    IF fRemDist < fPreTriggerPosition THEN
      eState             := cL_WAITSTART;
      tTrigger_EventTime := (tCurrentTime + LREAL_TO_ULINT(fRemDist / fI_ConveyorSpeed * 1E9));    // division save because we are moving to reach this position
      OnTriggerCommand   := cL_ACTIVE;  (*Arm EL2252*)

      LogTsDiff(aIdent := 'WAITALMOSTSTART: ', t1 := tTrigger_EventTime, t2 := tCurrentTime);
    ELSE
      eState           := cL_WAITALMOSTSTART;
      OnTriggerCommand := cL_INACTIVE;
    END_IF;

    ObTrigger := TRUE;

  cL_WAITSTART:       (*Wait until start time reached*)
    IF (tTrigger_EventTime < tCurrentTime) THEN (* StartTime elapsed *)
      // position reached
      eState           := cL_TRIGACTIVE;
      OnTriggerCommand := cL_INACTIVE; (*Disarm already command to EL2252, trigger generated*)
    ELSE
      // position not yet reached
      eState           := cL_WAITSTART;
      OnTriggerCommand := cL_ACTIVE;  (*Arm EL2252*)
    END_IF;

    ObTrigger := TRUE;  
    
  cL_TRIGACTIVE:   (*Trigger high*)
    eState := cL_WAITSTOP;
    
    // calculate end timestamp of trigger (end of trigger active signal)
    tTrigger_EventTime := (tTrigger_EventTime + LREAL_TO_ULINT(_fTriggerLength * 1E6));
    
    OnTriggerCommand := cL_INACTIVE;
    ObTrigger        := FALSE;
    
  cL_WAITSTOP:  (*Wait until trigger time has elapsed*)
    IF (tTrigger_EventTime < tCurrentTime) THEN (* StopTime elapsed *)
      eState           := cL_IDLE;
      OnTriggerCommand := cL_INACTIVE; (*Disarm EL2252, trigger generated*)
    ELSE
      eState           := cL_WAITSTOP;
      OnTriggerCommand := cL_ACTIVE;  (*Arm EL2252*)
    END_IF;

    ObTrigger        := FALSE;

  ELSE  (*Default*)
    eState           := cL_IDLE;
    ObTrigger        := FALSE;
    OnTriggerCommand := cL_INACTIVE;
END_CASE;

OtTriggerStartTime := tTrigger_EventTime;

(********************************* END OF FB *****************************************************)

METHOD Init
VAR_INPUT
  nResolution                   : LREAL := 1;      (*Printhead Resolution [e.g. 600] x Subpixel Resolution [e.g. 32]*)
  bUsePositionTrigger           : BOOL;            (*FALSE: Calculate time with speed and position distance@sensor evont*)
END_VAR
(*zero divisions*)
IF nResolution = 0 THEN RETURN; LogError('Invalid parameter'); END_IF;

// save config
_nResolution         := nResolution;
_bUsePositionTrigger := bUsePositionTrigger;

bInitOk := TRUE;
END_METHOD

(*
  Log timestamp difference (if verbose active).
  t1-t2 
*)
METHOD LogTsDiff : BOOL
VAR_INPUT
  aIdent : STRING;
  t1 : T_DCTIME64;
  t2 : T_DCTIME64;
END_VAR
IF _bVerbose THEN
  LogLvl(Lvl:=E_LogSeverity.Debug, Msg:=
       F_Concat7(aIdent, 
                 't1: ', TO_STRING(t1), 
                 ' t2: ', TO_STRING(t2), 
                 ' t1-t2 [ms]: ', TO_STRING((TO_LREAL(t1)-TO_LREAL(t2))*1E-6)
       )
  );
END_IF
END_METHOD

(*
  Detected start position X0 (absolute) in [SubPx].
*)
PROPERTY nStartPositionX0 : DINT
GET
nStartPositionX0 := _nX0;
END_GET
END_PROPERTY

PROPERTY UsePositionTrigger : BOOL
GET
UsePositionTrigger := _bUsePositionTrigger;
END_GET
SET
_bUsePositionTrigger := UsePositionTrigger;
END_SET
END_PROPERTY

END_FUNCTION_BLOCK

// ---- POUs/Products/FB_ModuleSynchronisation.TcPOU
FUNCTION_BLOCK FB_ModuleSynchronisation
VAR_INPUT
  IbEnable              : BOOL;             (*enable funcion*)
  IbEngaged             : ARRAY [1..iCPr_NB_PM] OF BOOL;
  IbPrintEnabled        : ARRAY [1..iCPr_NB_PM] OF BOOL;
  InFormatLength        : DINT;             (*format length [µm]*)
  InModule2ToModule3    : DINT;             (*distance between Module 2 and 3 [µm]*)
  IbFormatTrig          : BOOL;             (*format trigger*)
END_VAR

VAR_OUTPUT
  ObPrintEnabled        : ARRAY [1..iCPr_NB_PM] OF BOOL;
END_VAR

VAR
  fb_RFTrigPrintEnabled : RF_TRIG;
  fb_RTrigFormatTrig    : R_TRIG;
  _FormatTrigDelay      : DINT;             (*format trigger delay*)
  _FormatTrigCounter    : DINT;             (*format trigger counter*)
END_VAR

(*To start and stop printing of both modules synchronical the ObPrintEnabled of the second module must be delayed.*)
IF NOT IbEnable THEN
  ObPrintEnabled[1] := IbPrintEnabled[1];
  ObPrintEnabled[2] := IbPrintEnabled[2];
  RETURN;
END_IF

(*Trigger delay calculation*)
IF InFormatLength <> 0 THEN
  _FormatTrigDelay := InModule2ToModule3 / InFormatLength;
ELSE
  _FormatTrigDelay := 0;
END_IF

IF IbEngaged[1] THEN   (*Module2 active*)
  ObPrintEnabled[1] := IbPrintEnabled[1];   (*Module2 will print directly*)
  fb_RFTrigPrintEnabled(CLK := IbPrintEnabled[1]);
  IF fb_RFTrigPrintEnabled.RT THEN  (*Print start*)
    _FormatTrigCounter := 0;
    ObPrintEnabled[2] := FALSE;
  END_IF
  IF fb_RFTrigPrintEnabled.FT THEN  (*Print stop*)
    _FormatTrigCounter := 0;
  END_IF
  fb_RTrigFormatTrig(CLK := IbFormatTrig);
  IF fb_RTrigFormatTrig.Q THEN
    _FormatTrigCounter := _FormatTrigCounter + 1;
  END_IF
  IF _FormatTrigCounter >= _FormatTrigDelay THEN
    ObPrintEnabled[2] := IbPrintEnabled[2];     (*Module3 print is delayed*)
  END_IF
ELSE   (*Module3 can print directly*)
  ObPrintEnabled[1] := IbPrintEnabled[1];
  ObPrintEnabled[2] := IbPrintEnabled[2];
END_IF

END_FUNCTION_BLOCK

// ---- POUs/Products/obsolete/FB_CountWeu.TcPOU
FUNCTION_BLOCK FB_CountWeu
(*************************************************************************************************)
(*  FILENAME:    FB_CountWeu                                                                     *)
(*  PROJECT:     CALMAR PUPLC                                                                    *)
(*  COPYRIGHT:   All rights reserved (c) Wifag//Polytype, Fribourg/Switzerland (2021)            *)
(*  ENVIRONMENT: TwinCAT PLC                                                                     *)
(*  VERSION:     <version>                                                                       *)
(*************************************************************************************************)
(*  DESCRIPTION:                                                                   <description> *)
(*    Function for product count.                                                                *)
(*    The used pointers must be set in PRG_PRINT.Init!                                           *)
(*                                                                                </description> *)
(*************************************************************************************************)

VAR_INPUT
  pI_sAdsPrintUnit                          : POINTER TO ST_ADS_PU;        (*Pointer to ST_ADS_PU*)
  pI_ZeroPointerErr                         : POINTER TO UDINT;

  bI_SuccessFeedback                        : BOOL;             (*Success feedback from machine*)

  cI_ExtraCount                             : BYTE := 0;        (*Number of extra products that should be printed*)
END_VAR

VAR_OUTPUT
  bO_JobFinished                            : BOOL := FALSE;    (*Number of printed copies reached => job finished*)
  lO_ProductCountSuccess                    : UDINT;            (*Product counter of successfully printed*)
END_VAR

VAR
  iL_Counter                                : INT;              (*Local iteration counter - default*)

  lL_SuccessCount                           : UDINT := 0;       (*Success counter*)

  fb_RTrigSuccessFeedback                   : R_TRIG;           (*Success feedback from machine*)
  fb_RTrigPrintedCopies                     : R_TRIG;           (*Number of printed copies reached*)
END_VAR

(*0 pointer found*)
IF (pI_sAdsPrintUnit = 0) THEN
  IF pI_ZeroPointerErr <> 0 THEN
    pI_ZeroPointerErr^ := pI_ZeroPointerErr^ + 1;
  END_IF

  RETURN;
END_IF;

IF pI_sAdsPrintUnit^.sI_Start.bI_Command THEN
  lL_SuccessCount := 0;
END_IF;

(*Count successfull products*)
fb_RTrigSuccessFeedback(CLK := bI_SuccessFeedback);
IF fb_RTrigSuccessFeedback.Q THEN
  lL_SuccessCount := lL_SuccessCount + 1;
END_IF;
lO_ProductCountSuccess := lL_SuccessCount;

IF pI_sAdsPrintUnit^.sI_JobSettings.lI_NumberOfCopies = 0 THEN
  bO_JobFinished := FALSE;
ELSE
  (*Set job finished if number of desired copies reached.*)
  fb_RTrigPrintedCopies(CLK := (lL_SuccessCount >= (pI_sAdsPrintUnit^.sI_JobSettings.lI_NumberOfCopies + cI_ExtraCount)));
  IF fb_RTrigPrintedCopies.Q THEN
    bO_JobFinished := TRUE;
  END_IF;
END_IF;

(*Reset signals*)
IF pI_sAdsPrintUnit^.sI_Stop.bI_Command THEN
  bO_JobFinished := FALSE;
END_IF;

(********************************* END OF FB *****************************************************)

END_FUNCTION_BLOCK

// ---- POUs/Products/obsolete/FB_FIFO_DINT.TcPOU
FUNCTION_BLOCK FB_FIFO_DINT
(*************************************************************************************************)
(*  FILENAME:    FB_FIFO_TRIGGER_POS                                                             *)
(*  PROJECT:     CALMAR PUPLC                                                                    *)
(*  COPYRIGHT:   All rights reserved (c) Wifag//Polytype, Fribourg/Switzerland (2016)            *)
(*  ENVIRONMENT: TwinCAT PLC                                                                     *)
(*  VERSION:     <version>                                                                       *)
(*************************************************************************************************)
(*  DESCRIPTION:                                                                   <description> *)
(*    FIFO for trigger positions.                                                                *)
(*                                                                                </description> *)
(*************************************************************************************************)

{library public}
VAR_INPUT
  nI_FIFO_Input           : DINT;                          (*FIFO input value*)
  bI_Init                 : BOOL;                          (*Init*)
  bI_Add                  : BOOL;                          (*Add value*)
  bI_Release              : BOOL;                          (*Release value*)
END_VAR

VAR_OUTPUT
  bO_FIFO_Error           : BOOL;                          (*value FIFO error*)
  nO_FIFO                 : DINT;                          (*FIFO for value*)
END_VAR

{library private}
VAR
  nL_FIFO                 : ARRAY[0..iL_FIFOSIZE] OF DINT; (*FIFO for values*)
  iL_FIFO_Level           : INT := 0;                      (*Level of FIFO*)
  iL_Count                : INT;                           (*Temporary counter*)

  bL_Add                  : BOOL;                          (*Add value memory*)
  bL_Release              : BOOL;                          (*Release value memory*)
END_VAR

VAR CONSTANT
  (*Bit selection for configuration*)
  iL_FIFOSIZE             : INT := 75;
END_VAR

IF bI_Init THEN
  Init();
END_IF;

IF bI_Add AND NOT bL_Add THEN
  AddValue();
END_IF;
bL_Add := bI_Add;

IF bI_Release AND NOT bL_Release THEN
  ReleaseValue();
END_IF;
bL_Release := bI_Release;

nO_FIFO := nL_FIFO[0];
(********************************* END OF FB *****************************************************)

ACTION AddValue:
IF iL_FIFO_Level < iL_FIFOSIZE THEN
	nL_FIFO[iL_FIFO_Level] := nI_FIFO_Input;

	iL_FIFO_Level := iL_FIFO_Level + 1;
ELSE
	bO_FIFO_Error := TRUE;
END_IF;

(********************************* END OF ACTION *************************************************)
END_ACTION

ACTION Init:
iL_FIFO_Level := 0;
nL_FIFO[0]    := 0;
bO_FIFO_Error := FALSE;
(********************************* END OF ACTION *************************************************)
END_ACTION

ACTION ReleaseValue:
IF iL_FIFO_Level > 1 THEN
	FOR iL_Count := 0 TO (iL_FIFO_Level - 2) DO
		nL_FIFO[iL_Count] := nL_FIFO[iL_Count + 1];
	END_FOR;

	iL_FIFO_Level := iL_FIFO_Level - 1;
ELSIF iL_FIFO_Level = 1 THEN
	iL_FIFO_Level := 0;
END_IF;

(********************************* END OF ACTION *************************************************)
END_ACTION

END_FUNCTION_BLOCK

// ---- POUs/Products/obsolete/FB_HWLATCH.TcPOU
(* $Id$ *)
FUNCTION_BLOCK FB_HWLATCH
(*************************************************************************************************)
(*  FILENAME:     FB_HWLATCH.EXP			                                           		       		   *)
(*  PROJECT:      CALMAR PUPLC        																													 *)
(*  COPYRIGHT:    All rights reserved (c) Wifag//Polytype, Fribourg/Switzerland (2016)           *)
(*  ENVIRONMENT: 	TwinCAT PLC / CoDeSys																													 *)
(*	VERSION:			<version>																																			 *)
(*************************************************************************************************)
(*  DESCRIPTION:  Function block to convert hardware latch value [count] from terminal to print  *)
(*								system subpixel																																 *)
(*																																															 *)
(*************************************************************************************************)

{library public}
VAR_INPUT
	lI_Reference				:	UDINT;			(*position reference pulse count in [count]*)
	lI_Latch						:	UDINT;			(*position latch pulse count in [count]*)
	lI_Master_Position  :	DINT;				(*Current Master Position in [SubPx]*)
	fI_ResolutionInput	: LREAL:=1;	  (*Encoder Resolution in [um/increment]*)
	fI_ResolutionOutput	: LREAL:=1;	  (*Print system Resolution in [SubPx]*)
	bI_LatCVal					: BOOL;
	bI_Reset						: BOOL;				(*Reset terminal*)
END_VAR

VAR_OUTPUT
	iO_Offset_X0				: DINT;
	iO_Offset_XS				: DINT;
	bO_StartTrig				: BOOL;
	bO_EnLatC           : BOOL; 			(*C-Latch enable/reset @EL5101*)
END_VAR

{library private}
VAR
	lL_Latch_Reg				:	UDINT:=0;
  ll_Test             : UDINT:=0;
END_VAR

(*Latch register used for HW Start*)
IF lI_Latch <> lL_Latch_Reg AND bI_LatCVal THEN
  ll_Test := lI_Latch - lL_Latch_Reg;
	lL_Latch_Reg := lI_Latch;
	iO_Offset_X0 := lI_Master_Position - FC_LREAL_TO_DINT( (DINT_TO_LREAL(UDINT_TO_DINT(lI_Reference - lI_Latch)) * fI_ResolutionInput * (fI_ResolutionOutput / 25400) ));
	bO_StartTrig := TRUE;
ELSE
	bO_StartTrig := FALSE;
END_IF

(*Latch Handshake with Terminal EL5101,EnLatC must be set to 0 to reactivate latch input *)
IF bI_LatCVal THEN
	bO_EnLatC := FALSE;
ELSE
	bO_EnLatC := NOT bI_Reset;
END_IF

END_FUNCTION_BLOCK

// ---- POUs/Products/obsolete/FB_StartPositionDummy_HOA.TcPOU
(*
  A start position detection function block dummy.
  A dummy implementation to simulate start triggers at desired positions.
*)
FUNCTION_BLOCK FB_StartPositionDummy_HOA EXTENDS FB_BasePrint IMPLEMENTS I_StartPosDetect, I_PrintStatusClient, I_Simulation
VAR_INPUT
  bTrigger              AT%I* : BOOL;       // (INPUT) trigger (rising edge)
  tTrigger_TimeStamp    AT%I* : T_DCTIME64; // (INPUT) rigger timerstamp
  lPositionM2                 : DINT;       // current position [SubPx]
  fSpeedM2                    : LREAL;      // current speed [m/s]
  lPositionM3                 : DINT;       // current position [SubPx]
  fSpeedM3                    : LREAL;      // current speed [m/s]
  fResolution                 : LREAL;      // current print resolution [dpi*SubPx]
  nDelayTriggerDistance       : DINT;       // distance between CreateTrigger and DelayTrigger [SubPx]
  bMachineProdSpeed           : BOOL;       // machine reached production speed
  IpFormatLength              : POINTER TO DINT;  //pointer to format length if it's not used from iJobDefinition [µm]
END_VAR

VAR
  _bSim                 : BOOL;       // simulatio mode active (PROPERTY)
  _bCreateTrigger       : BOOL;       // create new CT trigger (PROPERTY)
  _nStartPosition       : DINT;       // create position for CT (absolut) [SubPx] (PROPERTY)
  _bCreateTriggerDelay  : BOOL;       // create delayed trigger (PROPERTY)
  _nDelayStartPosition  : DINT;       // create position for CT (absolut) [SubPx] (PROPERTY)
  fb_FIFOPositions      : FB_FIFO_DINT;
  _nFIFOPositionReg     : DINT;       // FIFO position register [SubPx]
  
  // local helper
  bNewCt              : BOOL;
  tCycle              : TIME;
  tonNewSheet         : TON;
  rfTrig_NewCT        : RF_TRIG;
  rfTrig_TriggerDelay : RF_TRIG;
  iJobDefinition      : CalmarCompPrint.I_JobDefinition;
  nCalcPosition       : DINT;            (*calculated position [SubPx]*)
  nCalcPositionM3     : DINT;            (*calculated position module 3 [SubPx]*)
  nDeltaPosition      : DINT;            (*delta position [SubPx]*)
  nDeltaPositionDelay : DINT;            (*delta position [SubPx]*)
  nSheetEndPosition   : DINT;            (*sheet end position [SubPx]*)
  nPositionRegM2      : DINT;            (*register position module 2 [SubPx]*)
  nPositionRegM3      : DINT;            (*register position module 3 [SubPx]*)
  nTriggerDistance    : DINT;            (*trigger distance [SubPx]*)
  bStartTrigger       : BOOL;            (*start trigger*)
  bSimStartTrigger    : BOOL;            (*simulated start trigger*)
  bSimStartActive     : BOOL;            (*simulated start active*)
  bInhibSensor        : BOOL;            (*inhibit sensor signals, TRUE=inhibit*)
  tCurrentTimeStamp   : T_DCTIME64;      (*get current timestamp*)
  fCurrentTimeStamp   : LREAL;           (*current timestamp*)
  fSensorTimeStamp    : LREAL;           (*sensor timestamp*)
  fDeltaDistance      : LREAL;           (*distance that the substrate moved between the detection and the treatment of the information [m]*)
END_VAR

VAR PERSISTENT
  // local simulation configurations persistent
  iCreateType    : UINT := 3;   // 0,1=by input rising edge, 2=create by sheets p.m. 3=create by sheet gap  
  fSheetCycle    : REAL := 20;  // [-] sheets per minute
  fSheetGap      : REAL := 0;   // [mm] gap between two sheets
  fSheetLength   : LREAL := 500; // [mm] sheet length TODO: remove if given by job(default if not given by jobDefinition)
END_VAR

VAR CONSTANT
  sCreateTArray : ARRAY[1..3] OF STRING := ['Input Trigger', 'Cycle', 'Gap'];
END_VAR

// Create CT triggers with a given cycle (based on configuration of Simulation)

(*If Module2 is disabled copy position from Module3*)
IF lPositionM2 = 0 THEN
  lPositionM2 := lPositionM3;
END_IF
(*Set nDelayTriggerDistance to minimum of 2 * IpFormatLength*)
IF (nDelayTriggerDistance <= LREAL_TO_DINT(F_SubPixelToMeter(2 * IpFormatLength^, fResSubPx := fResolution) * 1_000_000)) THEN 
  nDelayTriggerDistance := LREAL_TO_DINT(F_SubPixelToMeter(2 * IpFormatLength^, fResSubPx := fResolution) * 1_000_000);
END_IF


IF    iCreateType = 0 OR iCreateType = 1 OR NOT _bSim THEN   
  // --> trigger by input (default)
  IF bTrigger AND NOT bInhibSensor THEN
    bStartTrigger := TRUE;
    bInhibSensor  := TRUE;

    (* Calculate the current and sensor time stamp *)
    tCurrentTimeStamp := F_GetCurDcTaskTime64();
    fCurrentTimeStamp := (ULINT_TO_LREAL(tCurrentTimeStamp )) / 1_000_000.0; (*in ms*)
    fSensorTimeStamp  := fCurrentTimeStamp;// (ULINT_TO_LREAL(tTrigger_TimeStamp)) / 1_000_000.0; (*in ms*)
    (* Treatment of the information *)
    fDeltaDistance := (fCurrentTimeStamp - fSensorTimeStamp) * 0.001 * fSpeedM2;  (*Distance that the substrate moved between the detection and the treatment of the information [m]*)
    nCalcPosition     := lPositionM2 - F_MeterToSubPixel(fPosMeter := fDeltaDistance, fResoSubPx := fResolution);
    nSheetEndPosition := nCalcPosition + F_MeterToSubPixel(fPosMeter := fSheetLength / 1000, fResoSubPx := fResolution);
  ELSE
    bStartTrigger := FALSE;
	END_IF

  bNewCt := bStartTrigger;

ELSIF iCreateType = 2 AND _bSim THEN   
  // --> trigger by sheets per minute
  tCycle := prodspeed_to_time(lCycle := fSheetCycle);
  tonNewSheet(IN := NOT tonNewSheet.Q, PT := tCycle, Q => bNewCt);
  nCalcPosition := lPositionM2;
  
ELSIF iCreateType = 3 AND _bSim THEN
  // --> trigger by sheet gap;

  // fSheetLength from other source
  IF (IpFormatLength <> 0) THEN
    fSheetLength := DINT_TO_LREAL(IpFormatLength^) / 1000; // [µm] -> [mm]
  END_IF

  //  we need current job settings
  IF fSheetLength = 0 THEN fSheetLength := 1*1000; END_IF  // set some valid size 1000mm if no job is given
  (*trigger with timer is too inaccurate!*)
  (*
  IF (fSpeed > 0) THEN
    tCycle := length_to_time(dist := (fSheetGap + fSheetLength) / 1000, speed := fSpeed); 
    tonNewSheet(IN := NOT tonNewSheet.Q, PT := tCycle, Q => bNewCt);
  END_IF
  nCalcPosition := lPosition;
  *)

  (*trigger with distances*)
  bNewCt := FALSE;
  IF NOT bMachineProdSpeed THEN
    bSimStartActive  := FALSE;
  ELSE
    nTriggerDistance := F_MeterToSubPixel(fPosMeter := (fSheetGap + fSheetLength) / 1000, fResoSubPx := fResolution);

    IF NOT bSimStartActive THEN
      bSimStartActive     := TRUE;
      nDeltaPosition      := 0;
      nDeltaPositionDelay := 0;
      nPositionRegM2      := lPositionM2;
      nPositionRegM3      := lPositionM3;
		END_IF
    nDeltaPosition      := nDeltaPosition      + (lPositionM2 - nPositionRegM2);
    nDeltaPositionDelay := nDeltaPositionDelay + (lPositionM3 - nPositionRegM3);

    IF (nDeltaPosition >= nTriggerDistance) THEN
      bNewCt          := TRUE;
      nCalcPosition   := lPositionM2 - (nDeltaPosition - nTriggerDistance);
      nCalcPositionM3 := lPositionM3 - (nDeltaPosition - nTriggerDistance);
      nDeltaPosition  := nDeltaPosition - nTriggerDistance;
    END_IF
  END_IF
ELSE
  ;  // not supported ignore
END_IF


// Module 2: set ouputs (properties)
rfTrig_NewCT(CLK := bNewCt, RT => _bCreateTrigger);    // set ouput trigger
IF _bCreateTrigger THEN 
  _nStartPosition := nCalcPosition;
END_IF

// Module 3: set ouput for delay trigger (properties)
fb_FIFOPositions( bI_Init       := NOT bMachineProdSpeed  (*OR (nDelayTriggerDistance = 0)*)
                , bI_Add        := _bCreateTrigger
                , bI_Release    := _bCreateTriggerDelay
                , nI_FIFO_Input := nCalcPositionM3);
_nDelayStartPosition := fb_FIFOPositions.nO_FIFO + nDelayTriggerDistance;
IF _nFIFOPositionReg <> fb_FIFOPositions.nO_FIFO THEN
  nDeltaPositionDelay := (lPositionM3 - fb_FIFOPositions.nO_FIFO);
END_IF
_nFIFOPositionReg := fb_FIFOPositions.nO_FIFO;

rfTrig_TriggerDelay( CLK :=     (nDeltaPositionDelay >= nDelayTriggerDistance) 
                            AND bMachineProdSpeed
                            AND (fb_FIFOPositions.nO_FIFO <> 0)
                   , RT => _bCreateTriggerDelay);    // set ouput trigger


(*stop trigger to reset bInhibSensor*)
IF (lPositionM2 >= nSheetEndPosition) AND bInhibSensor THEN
  bInhibSensor := FALSE;
END_IF;

(*register position*)
nPositionRegM2 := lPositionM2;
nPositionRegM3 := lPositionM3;

PROPERTY bSimEnable : BOOL
GET
bSimEnable := _bSim;
END_GET
SET
_bSim := bSimEnable;
END_SET
END_PROPERTY

(*
  A new container detected.
  NOTE: a pulse only
*)
PROPERTY bStartTrig : BOOL
GET
bStartTrig := _bCreateTrigger;
END_GET
END_PROPERTY

(*
  A new container detected.
  NOTE: a pulse only
*)
PROPERTY bStartTrigDelay : BOOL
GET
bStartTrigDelay := _bCreateTriggerDelay;
END_GET
END_PROPERTY

(*
  A valid container detected.
*)
PROPERTY bValid : BOOL
GET
bValid := TRUE;
END_GET
END_PROPERTY

(*
Convert a distance to time with current speed
*)
METHOD PRIVATE length_to_time : TIME
VAR_INPUT
  dist  : LREAL; // [m] distance
  speed : LREAL; // [m/s] @speet
END_VAR
IF speed = 0 THEN  RETURN; END_IF   // ignore if speed = 0

length_to_time := LREAL_TO_TIME((dist * 1000)/ speed);  // TIME base is in [ms]
END_METHOD

METHOD mJobPause
END_METHOD

METHOD mJobStart
VAR_INPUT
	sJobDef	: CalmarCompPrint.I_JobDefinition;
END_VAR

// sample new CT configuration from job
iJobDefinition := sJobDef;    // current job definition

// fSheetLength from job definition
IF (iJobDefinition <> 0) AND (IpFormatLength = 0) THEN
  fSheetLength := iJobDefinition.fSubstrateDepth * 1000; // [m] -> [mm]
END_IF
// fSheetLength from other source
IF (IpFormatLength <> 0) THEN
  fSheetLength := DINT_TO_LREAL(IpFormatLength^) / 1000; // [µm] -> [mm]
END_IF

bInhibSensor := FALSE;
END_METHOD

METHOD mJobStop
VAR_INPUT
	sStatus	: CalmarCompPrint.I_JobStatus;
END_VAR
iJobDefinition := 0;    // delete job definition
END_METHOD

METHOD mProduced
VAR_INPUT
	(* current progress*)
	sProgress	: CalmarCompPrint.I_JobProgress;
END_VAR
; // nothing to do
END_METHOD

(*
  Detected start position X0 (absolute) in [SubPx].
*)
PROPERTY nDelayStartPositionX0 : DINT
GET
nDelayStartPositionX0 := _nDelayStartPosition;
END_GET
END_PROPERTY

(*
  Detected start position X0 (absolute) in [SubPx].
*)
PROPERTY nStartPositionX0 : DINT
GET
nStartPositionX0 := _nStartPosition;
END_GET
END_PROPERTY

(*
Convert production speed to a time. E.g. number of sheet per minute to a cycle time.
*)
METHOD PRIVATE prodspeed_to_time : TIME
VAR_INPUT
  lCycle        : REAL;    // sheets per minute
END_VAR
VAR
  fCycleTime    : LREAL;
END_VAR
fCycleTime := (60 / REAL_TO_LREAL(lCycle)) * 1000;
prodspeed_to_time := LREAL_TO_TIME(fCycleTime);
END_METHOD

METHOD reset
VAR_INPUT
END_VAR
bSimStartActive := FALSE;
END_METHOD

METHOD SimEnter : BOOL
LogInfo('Enter start position creator simulation');
_bSim := TRUE;
END_METHOD

METHOD SimExit : BOOL
LogInfo('Exit start position creator simulation');
_bSim := FALSE;
END_METHOD

METHOD SimUpdate : BOOL
; // nothing to do
END_METHOD

END_FUNCTION_BLOCK

// ---- POUs/Products/obsolete/FB_WorkerWeu.TcPOU
FUNCTION_BLOCK ABSTRACT FB_WorkerWeu EXTENDS FB_Worker
VAR_OUTPUT
  bError        : BOOL;       // an error is active
  nError        : UDINT;      // error code if error active, =0 else
END_VAR
VAR
  // config
  _pCtManager       : POINTER TO FB_CTManagerDefGrid;  // CT Manager reference
  _nTrackPosDomain  : E_PosDomain;    // Tracking position domain 
  _fPrintResolution : LREAL := 1;     // print(head) resolution in [dpi]
  _fSubPxResolution : LREAL := 1;     // SubPixel resolution [SubPx], resolution factor (fI_PrintResolution*fI_SubPxResolution=>Output resolution
  _name             : STRING;         // Worker name
  _sVisuName        : STRING := 'VISU_WorkerWeu'; // Worker visu instance name
  _pEcSrc           : POINTER TO T_ErrSrc;       // Error source definition

  // job
  _bJobActive       : BOOL;           // a job is active
  // ct
  _pAttachedCt      : POINTER TO FB_ContainerDefGrid;  // currently attached container
  fCtPosition       : LREAL;          // Container position relative to worker position in [SubPx (E_PosDomain.master_pos)]
  _bForceRelease    : BOOL;
END_VAR
VAR_STAT
  // static variables, same for all Workers
  _aJobName         : T_MaxString;
  _aJobGuid         : T_MaxString;
  _fImageWidthM     : LREAL;          // image width in [m]
  _fImageDepthM     : LREAL;          // image depth in [m]
  _fCtSecurityReleasePos : LREAL := 0;     // [SubPx] position where to release current ct at last (security release)
END_VAR
VAR PERSISTENT
  _fWorkerPosition  : LREAL;          // worker position relative to X0 in [m]
END_VAR

(*
  Generic abort implementation of DefGrid CT.
*)
METHOD Abort
VAR_INPUT
  iCT       : I_CT;
  sReason   : STRING;
END_VAR
VAR
  _pCt   : POINTER TO FB_ContainerWeu;
END_VAR
IF getCtInst(iCT:=iCT, pCT=>_pCt) <> 0 THEN  // get specific container
  // Do generic known aborts on CT
END_IF
END_METHOD

METHOD PROTECTED  Attach : BOOL
VAR_INPUT
  iCT       : I_CT;            (*container at triggered event position*)
END_VAR
VAR
  _pNewCt   : POINTER TO FB_ContainerWeu;

END_VAR
IF iCT = 0 THEN
  LogError(Msg:='attach failed -> not ct given');
  
ELSIF bEnable AND _pAttachedCt = 0 THEN           // enabled and free to attach
  IF getCtInst(iCT:=iCT, pCT=>_pNewCt) <> 0 THEN  // get specific container
    _pAttachedCt := _pNewCt;
    Attach:=TRUE;                                 // attach new
  ELSE
    LogError(Msg:='attach failed');
  END_IF
  
ELSIF bEnable AND _pAttachedCt <> 0 THEN    // enabled and already a CT attached
  LogError(Msg:='another container already attached -> ignore new (set error)');
  Abort(iCT:=iCT, sReason:='attach failed');  // abort new CT
    
ELSIF NOT bEnable AND _pAttachedCt <> 0 THEN // disabled and already a CT attached
  // force release if any hanging, and ignore attach
  Release(iCT:=_pAttachedCt^);

ELSIF NOT bEnable AND _pAttachedCt = 0 THEN  
  ;   // nothing to do, ignore attach

ELSE      // unspecified (error)case just log it
  LogError(Msg:='not tracked case');
END_IF
END_METHOD

{attribute 'monitoring':='call'}
PROPERTY bAttached : BOOL
GET
IF _pAttachedCt <> 0 THEN
  bAttached := TRUE;
END_IF
END_GET
END_PROPERTY

{attribute 'monitoring':='call'}
PROPERTY fPosition : LREAL
GET
fPosition := _fWorkerPosition;
END_GET
SET
_fWorkerPosition := fPosition;
setupPosition();
END_SET
END_PROPERTY

{attribute 'monitoring':='call'}
PROPERTY fPrintResolution : LREAL
GET
fPrintResolution := _fPrintResolution;
END_GET
SET
_fPrintResolution := fPrintResolution;
setupPosition();
END_SET
END_PROPERTY

(*
  Get specific container from interface.
  Returns specific container in return value and output parameter.
*)
METHOD INTERNAL getCtInst : POINTER TO FB_ContainerWeu
VAR_INPUT
  iCT              : I_CT;                         (*container at triggered event position*)
END_VAR
VAR_OUTPUT
  pCT              : POINTER TO FB_ContainerWeu;
END_VAR
pCT := 0;
IF _pCtManager <> 0 THEN
  getCtInst := _pCtManager^.GetContainerInstance(iCT);   // get real ct fb inst
  IF getCtInst <> 0 THEN
    pCT := getCtInst;   // OK all good
  ELSE
    LogError(Msg:='specific container not found');
	END_IF
ELSE
  LogError(Msg:='no container manager');
END_IF
END_METHOD

METHOD Init
VAR_INPUT
  pCtManager : POINTER TO FB_CTManagerWeu;       // CTManager
  fPrintResolution : LREAL := 1;                 // print(head) resolution in [dpi]
  fSubPxResolution : LREAL := 1;                 // SubPixel resolution [SubPx], resolution factor (fI_PrintResolution*fI_SubPxResolution=>Output resolution)
END_VAR
_pAttachedCt:=0;

IF pCtManager = 0 THEN
  LogError(Msg:='Init: invalid parameter');
  RETURN;
END_IF

// save config
_pCtManager := pCtManager; 
_fPrintResolution := fPrintResolution;
_fSubPxResolution := fSubPxResolution;
_fCtSecurityReleasePos := 0;
setupPosition();

setName('');

// register worker CTManager/Tracker event subject
_nTrackPosDomain := E_PosDomain.master_pos;
_pCtManager^.RegisterPosition(nPosDomain:=_nTrackPosDomain, iPositionEvent:=THIS^);

// init error source reference
_pEcSrc := ErrorCodes.fbErrCodeMngr.registerErrSource(
 nLocId := 0,
 aInstPath := InstanceName,
 aLocDescr := _name
);
IF _pEcSrc = 0 THEN LogError('could not register error source'); END_IF

bInitialized := TRUE;
END_METHOD

METHOD  ABSTRACT mJobStart
VAR_INPUT
	sJobDef	: CalmarCompPrint.I_JobDefinition;
END_VAR
END_METHOD

METHOD ABSTRACT mJobStop
VAR_INPUT
	sStatus	: CalmarCompPrint.I_JobStatus;
END_VAR
END_METHOD

(*
  Release CT from Worker.
  :return: TRUE if CT was released, FALSE if no CT was registered 
*)
METHOD Release : BOOL
VAR_INPUT
  iCT              : I_CT;                         (*container at triggered event position*)
END_VAR
IF iCT <> 0 AND _pAttachedCt <> 0 THEN Release := TRUE; END_IF
_pAttachedCt:=0;
END_METHOD

METHOD PRIVATE setName : BOOL
VAR_INPUT
  sName : STRING;
END_VAR
VAR
  nIdx : INT;
  bDone : BOOL;
END_VAR
IF sName = '' THEN
  // generate worker name
  _name := THIS^.InstanceName;
  WHILE NOT bDone DO
    nIdx := FIND(_name, '_');
    IF nIdx = 0 THEN bDone := TRUE; EXIT; 
    ELSE
      _name := RIGHT(_name,LEN(_name)-nIdx);
    END_IF 
  END_WHILE
ELSE
  _name := sName;  
END_IF
END_METHOD

METHOD PROTECTED setupPosition
_nTrackOffset := F_MeterToSubPixel(fPosMeter:=fPosition, fResoSubPx:=_fPrintResolution*_fSubPxResolution);
END_METHOD

METHOD  work
//Work only with attached container
IF _pAttachedCt <> 0 THEN 
  
  // update CT position
  fCtPosition := _pAttachedCt^.GetPos(nPosDomain:=E_PosDomain.master_pos) - _nTrackOffset; 

  // release CT (manually and security)
  IF _bForceRelease THEN
    LogWarning(F_Concat2('Manually realease CTId=', TO_STRING(_pAttachedCt^.pCT^.iId)));
    Release(iCT:=_pAttachedCt^);
  ELSIF _fCtSecurityReleasePos > 0 AND (fCtPosition > _fCtSecurityReleasePos) THEN
    LogError(F_Concat2('Security released CTId=', TO_STRING(_pAttachedCt^.pCT^.iId)));
    Release(iCT:=_pAttachedCt^);
  END_IF
  
END_IF
END_METHOD

END_FUNCTION_BLOCK

// ---- POUs/Products/obsolete/FB_WorkerWeu_Print.TcPOU
FUNCTION_BLOCK FB_WorkerWeu_Print EXTENDS FB_WorkerWeu
VAR_INPUT
  nEncoderPos   : DINT;       // Absolute print position [SubPx]
  fEncoderSpeed  : LREAL;     // Print speed [m/s]
  bHardwareSync : BOOL;
  bHardwareHold : BOOL;
  fPrintStartOffset : LREAL;  //PU->PG/PA offset
  fPrintYOffset : LREAL;      //Y-Shift in ram memory
END_VAR
VAR_OUTPUT
END_VAR
VAR
  fbPs              : FB_PS;
  fbPa              : FB_PA;
  fB_PcAdapter      : FB_PC_Adapter;
  
  _fPrintStartOffset : LREAL;   // internal print start offset
  _nPosX0            : DINT;    // X0 for last attached CT (detected postion)
  _nPosXS            : DINT;    // XS for last attached CT (shifted print start position)
  _nPosXDelta        : DINT;    // Shift value X0 -> XS
  _fPosY             : LREAL;    // Y shift for last attached CT
  _bPaStarted        : BOOL;
  _bPaStartRequested : BOOL;
  fBStartTimeout     : TON;
  rTrigSync          : R_TRIG;

  (*Messaging*)
  _bMsgInitialized   : BOOL;
  fb_MsgQueue        : FB_MSG_QUEUE;                        (*Message queue*)
  fb_MsgHandler      : FB_MSG_HANDLER;                      (*Message handler*)
  sL_MsgConfig       : ST_MSG_CONFIG;                       (*Message config*)
  fb_Msg             : ARRAY [1..iC_NUM_MSG] OF FB_MESSAGE; (*Messages*)
END_VAR
VAR PERSISTENT
  _fStartShiftOffset : LREAL := fC_START_SHIFT_OFFSET;
  _fStartShiftFactor : LREAL := fC_START_SHIFT_FACTOR;
END_VAR
VAR CONSTANT
  iC_NUM_MSG : UDINT := 5;
  fC_START_SHIFT_FACTOR : LREAL := -2.4E-2;
  fC_START_SHIFT_OFFSET : LREAL := -1.0E-2;
END_VAR


//TODO Add error/warnings
bError := FALSE;
nError := 0;

//Start offset update
IF _fPrintStartOffset <> fPrintStartOffset THEN //Worker position changed
  IF _pAttachedCt = 0 THEN //Update only without attached container
    _fPrintStartOffset :=fPrintStartOffset;
	END_IF
END_IF

//Worker position update
IF _fWorkerPosition <> (_fPrintStartOffset + (_fStartShiftOffset + _fStartShiftFactor * fEncoderSpeed))  THEN //Worker position changed (camera settings change)
  IF _pAttachedCt = 0 THEN //Update only without attached container
    // WorkerPosition
    fPosition := _fPrintStartOffset + (_fStartShiftOffset + _fStartShiftFactor * fEncoderSpeed);
	END_IF
END_IF

(*---- Messaging -----------------------*)
IF _bMsgInitialized THEN
  fb_MsgHandler();
  {warning 'TODO: implement PrintWorker & PG messages'}
  //fB_Msg[1](bI_Status := dfsdfdsf);
  fb_MsgQueue();
END_IF

PROPERTY aPaState : STRING
GET
aPaState := fbPa.aPaState;
END_GET
END_PROPERTY

METHOD PROTECTED  Attach : BOOL
VAR_INPUT
  iCT              : I_CT;                         (*container at triggered event position*)
END_VAR
Attach:=FALSE;

IF bEnable AND SUPER^.Attach(iCT:=iCT) THEN
  // Additional worker checks
    // - job is valid?
  IF _pAttachedCt^.pJob = 0 OR NOT _bJobActive THEN
    Release(iCT:=iCT);
    RETURN;   // do not print
  
  // CT valid & CT present
  ELSIF NOT _pAttachedCt^.bValid OR NOT _pAttachedCt^.bProductPresent THEN
    Release(iCT:=iCT);
    RETURN;   // do not print
  
  // Ignore start due to hardware hold  
  ELSIF bHardwareHold THEN
    //_pAttachedCt^.setError(ErrDef:=EC_Print.ecPaAbortHold, Src:=_pEcSrc^);
    Release(iCT:=iCT);
    RETURN;   // do not print
  // - OK attach
  ELSE
    Attach := TRUE;
	END_IF
  
  
  //Prepare print station
  fbPs.bPrintEnable := iCT.bValid AND iCT.bProductPresent;

  //Start print, PA should be in READY or DONE
  
  // Set X print position
  _nPosX0 := _pAttachedCt^.getPosX0(nPosDomain:=E_PosDomain.master_pos);
  _nPosXDelta := F_MeterToSubPixel(_fPrintStartOffset,_fPrintResolution*_fSubPxResolution); // + PG/PA Shift (additional PG offset 0 for firstLine)

  _nPosXS := _nPosX0 + _nPosXDelta;
  fB_PcAdapter.setPrintStartPos(nX0:=_nPosXS);
  
  // Set Y print position
  _fPosY := fPrintYOffset;
  fB_PcAdapter.setPrintYShift(nYShift:=FC_LREAL_TO_DINT(_fPosY));

  // check
  IF _nPosXS < nEncoderPos THEN
    LogWarning(Msg:='Print start position < Encoder position');
	END_IF
    
  IF fbPa.printStart() THEN
    _bPaStarted := FALSE;
    _bPaStartRequested := TRUE;
    Attach:=TRUE;
    LogLvl(Lvl:=E_LogSeverity.Debug, F_Concat2('printStart:', _pAttachedCt^.print(0)));  // print container
    LogLvl(Lvl:=E_LogSeverity.Debug, F_Concat4('> XS:', TO_STRING(_nPosXS), ' = X0:', TO_STRING(_pAttachedCt^.GetPosX0(nPosDomain:=E_PosDomain.master_pos))));
    LogLvl(Lvl:=E_LogSeverity.Debug, F_Concat2( ' + shStartOffs:', TO_STRING(F_MeterToSubPixel(_fPrintStartOffset,_fPrintResolution*_fSubPxResolution))));

  ELSE  
    LogError(Msg:='PA not ready to start at attach');
    Release(iCT := iCT);
	END_IF
  
ELSE
  // parent attach failed case
END_IF
END_METHOD

METHOD InitMsg : BOOL
VAR_INPUT
  pMsgInterface : POINTER TO ST_ADS_MSG_IF;
END_VAR
VAR
  nCtr : UDINT;
END_VAR
IF pMsgInterface = 0 THEN RETURN; END_IF

(*Messaging*)
sL_MsgConfig.bI_Enable       := TRUE;
sL_MsgConfig.pI_FbMsgHandler := ADR(fb_MsgHandler);
fb_MsgHandler.pI_MsgQueue    := ADR(fb_MsgQueue);
fb_MsgQueue.pI_MsgInterface  := pMsgInterface;
fb_MsgQueue.cI_MaxElement    := 6;

(*Messages*)
FOR nCtr := 1 TO iC_NUM_MSG DO
  fb_Msg[nCtr].pI_MsgConfig       := ADR(sL_MsgConfig);
  fb_Msg[nCtr].iI_MsgLocation     := 0;
END_FOR
//fb_Msg[1].iI_MsgNumber       := ;
// ...

_bMsgInitialized := TRUE;
END_METHOD

METHOD InitWorkerPrint : BOOL
VAR_INPUT
END_VAR
IF NOT bInitialized THEN LogError('Base Worker not initialized! call init() before'); RETURN; END_IF

// worker specific init

//Print Aggregate
fbPa.bSyncAfterDone := FALSE;
fbPa.init(iPcAdapter := fB_PcAdapter, iPsInterface:=fbPs);
END_METHOD

METHOD   mJobStart
VAR_INPUT
	sJobDef	: CalmarCompPrint.I_JobDefinition;
END_VAR
IF NOT bEnable THEN RETURN; END_IF  // only if enabled

fbPa.jobStart();

_bJobActive := TRUE;
END_METHOD

METHOD  mJobStop
VAR_INPUT
	sStatus	: CalmarCompPrint.I_JobStatus;
END_VAR
fbPa.jobStop();
_bJobActive := FALSE;
END_METHOD

METHOD registerPc : BOOL
VAR_INPUT
  iNewPC : I_PC;
END_VAR
registerPc := fB_PcAdapter.registerPc(iNewPC := iNewPC);
END_METHOD

METHOD registerPh : BOOL
VAR_INPUT
    iPH : I_PH;
END_VAR
//Attach head to print station
IF iPH <> 0 THEN
  fbPs.registerPh(iNewPh:=iPH);
END_IF
END_METHOD

PROPERTY sPcFlags : CalmarCompPrint.ST_PC_FLAGS
GET
sPcFlags := fB_PcAdapter.sPcFlags;
END_GET
END_PROPERTY

PROPERTY sPcState :  CalmarCompPrint.ST_PG_STATUS
GET
VAR
  sJobStatus : ST_JobProgress;
END_VAR
sPcState.bStartPrintCanEx := fBPa.bStartCanEx;
sPcState.bStartPrintExec  := fBPa.bStartExec;
sPcState.bStopPrintCanEx  := fBPa.bStopCanEx;
sPcState.bStopPrintExec   := fBPa.bStopExec;
sPcState.bPausePrintCanEx := FALSE;       // obsolete ???
sPcState.bPausePrintExec  := FALSE;       // obsolete ???
sPcState.bReady           := fB_PcAdapter.bAllReady OR fB_PcAdapter.bAllDone;
sPcState.bError           := fB_PcAdapter.bError;
sPcState.bPrinting        := fB_PcAdapter.bAllPrinting;
sPcState.bLoad            := fB_PcAdapter.bAllPreparing;
sPcState.bArmed           := fB_PcAdapter.bAllPrinting OR fB_PcAdapter.bAllReady OR fB_PcAdapter.bAllDone OR fB_PcAdapter.bAllPreparing;
sPcState.bEnabled         := bEnable;
sPcState.bStartStrb       := fBPa.bStartStrb;
sPcState.bPcEnabled       := fB_PcAdapter.bPcEnable;
sPcState.lProductCount    := 0;            // obsolete ???
sPcState.sJobStatus       := sJobStatus;   // obsolete ???
END_GET
END_PROPERTY

METHOD  work
IF NOT bEnable THEN RETURN; END_IF

SUPER^.work();

(*Update virtual encoder on all controller boards*)
fB_PcAdapter.setEncoderPos(nEncoderPos);
fB_PcAdapter();

(*Call print aggregate*)
rTrigSync(CLK:=bHardwareSync); 
IF rTrigSync.Q THEN fbPa.sync(); END_IF   // external sync
fbPa.bHold := bHardwareHold;              // external hw hold
fbPa();

fBStartTimeout(IN := _bPaStartRequested,PT := T#60MS);

IF _pAttachedCt <> 0 AND bEnable THEN // Work only with attached container
  // PA control
  IF bHardwareHold THEN   // _pAttachedCt^.bValid AND
    // abort during printing
    _pAttachedCt^.setError(ErrDef:=EC_Print.ecPaAbortHold, Src:=_pEcSrc^);
    Release(_pAttachedCt^);
    
  ELSIF _bPaStartRequested THEN
    IF fbPa.bPrinting THEN
      _bPaStarted := TRUE;
      _bPaStartRequested := FALSE;
    ELSIF fBStartTimeout.Q THEN //Stop print at timeout to make ready for next container
      _bPaStarted := FALSE;
      _bPaStartRequested := FALSE;
      fbPa.printStop();
      _pAttachedCt^.setError(ErrDef:=EC_Print.ecPaStartErr, Src:=_pEcSrc^);
      Release(_pAttachedCt^);
		END_IF
  ELSIF _bPaStarted THEN
    // Set Y print position
    _fPosY := fPrintYOffset;
    fB_PcAdapter.setPrintYShift(nYShift := FC_LREAL_TO_DINT(_fPosY));

    //Release container when print finished
    IF fbPa.bDone OR fbPa.bStop THEN
      _bPaStarted := FALSE;
      Release(_pAttachedCt^);
    (*ELSIF fbpa.bError THEN
      _pAttachedCt^.setError(ErrDef:=EC_Print.ecPaPrintErr, Ident:=0);
      Release(_pAttachedCt^);*)
    END_IF 
	END_IF
END_IF  

(*Logging config*)
fbPa.LogLevel := LogLevel;
fB_PcAdapter.LogLevel := LogLevel;
END_METHOD

END_FUNCTION_BLOCK

// ---- POUs/Products/Print_Weu/UV_LED_Modul/FB_UvLedModule.TcPOU
FUNCTION_BLOCK FB_UvLedModule EXTENDS FB_BasePrint IMPLEMENTS I_DeviceBase
VAR_INPUT
  IbReady                  AT%I* : BOOL;
END_VAR

VAR_OUTPUT
  ObEnableHigh             AT%Q* : BOOL;
  ObLowIntenseMode         AT%Q* : BOOL;
  ObDisableLeft            AT%Q* : BOOL;
  ObDisableRight           AT%Q* : BOOL;
  OnIntensitySetpoint      AT%Q* : WORD;  (*Setpoint for intensity control  [digit]*)
END_VAR

VAR
  _bActivate                     : BOOL;
  _sName                         : STRING := '';
  _StInkDefinition               : ST_INKDEFINITON;
END_VAR

VAR CONSTANT
  CnAnalogMinDigit               : DINT := 0;      (*Min value analog-output in digit*)
  CnAnalogMaxDigit               : DINT := 32767;  (*Max value analog-output in digit*)
  CnMinIntensitySetpoint         : DINT := 5;      (*Min setpoint for intensity control [%]*)
  CnMaxIntensitySetpoint         : DINT := 100;    (*Max setpoint for intensity control [%]*)
END_VAR

VAR PERSISTENT
  RbLowIntenseMode               : BOOL := FALSE;  (*Visu: set low intense mode*)
  RbDisableLeft                  : BOOL := FALSE;  (*Visu: disable left SLM*)
  RbDisableRight                 : BOOL := FALSE;  (*Visu: disable right SLM*)
  RnIntensitySetpoint            : DINT := 20;     (*Visu: setpoint for intensity control [%]*)
END_VAR

(*Set outputs*)
ObEnableHigh        := _bActivate;
ObLowIntenseMode    := RbLowIntenseMode;
ObDisableLeft       := RbDisableLeft;
ObDisableRight      := RbDisableRight;
OnIntensitySetpoint := DINT_TO_WORD(CnAnalogMaxDigit * RnIntensitySetpoint / 100);  (*Setpoint [digit]*)

METHOD mDisable : BOOL
_bActivate := FALSE;
END_METHOD

METHOD mEnable : BOOL
_bActivate := TRUE;
END_METHOD

{warning 'add property implementation'}
PROPERTY pActive : BOOL
GET
pActive := _bActivate;
END_GET
END_PROPERTY

{warning 'add property implementation'}
PROPERTY pErrorCode : INT
GET
END_GET
END_PROPERTY

PROPERTY pStInkDefinition : ST_INKDEFINITON
SET
_StInkDefinition := pStInkDefinition;
END_SET
END_PROPERTY

END_FUNCTION_BLOCK

// ---- Project Information/F_GetCompany.TcPOU
// This function has been automatically generated from the project information.
{attribute 'signature_flag' := '1073741824'}
{attribute 'TcGenerated'}
{attribute 'no-analysis'}
FUNCTION F_GetCompany : WSTRING
VAR_INPUT
	
END_VAR

F_GetCompany := "WIFAG-Polytype";

END_FUNCTION

// ---- Project Information/F_GetTitle.TcPOU
// This function has been automatically generated from the project information.
{attribute 'signature_flag' := '1073741824'}
{attribute 'TcGenerated'}
{attribute 'no-analysis'}
FUNCTION F_GetTitle : WSTRING
VAR_INPUT
	
END_VAR

F_GetTitle := "PUPLC";

END_FUNCTION

// ---- GlobalTextList.TcGTLO
TEXTLIST GlobalTextList
  469 = ' '
  412 = '  %d'
  419 = '  %s'
  415 = '  0x%X'
  585 = '  1     2    3     4    5     6    7    8'
  295 = '  :'
  13539 = '  > verbose Mode'
  10089 = '  Delta distance [m]: %f'
  818 = '  Dropspeed [m/s]: %f'
  13004 = '  Module for mark trigger: %d'
  16821 = '  Time distance [ms]: %d'
  782 = ' %f'
  7576 = ' %s'
  10973 = ' %s ID'
  10174 = ' (max %d)'
  24 = ' ActualLevel'
  2816 = ' Add. dead time [ms]: %f'
  476 = ' Base folder: %s'
  990 = ' Camera correction X [m]: %f'
  987 = ' Camera correction [m]: %f'
  781 = ' Camera offset Y [mm]: %f'
  772 = ' Camera position X [m]: %f'
  831 = ' Camera position [m]: %f'
  471 = ' CH0: %d %%'
  472 = ' CH1: %d %%'
  473 = ' CH2: %d %%'
  474 = ' CH3: %d %%'
  820 = ' Compensation [mm]: %f'
  828 = ' Current time stamp compensation [µs]: %d'
  489 = ' D: %d'
  4 = ' ErrorLevel'
  492 = ' FileNbrs : %d '
  493 = ' Files p. PC : %d '
  5911 = ' Head base plate gap to roller table [m]: %f'
  1154 = ' Head offset to base plate [m]: %f'
  484 = ' ID: %d'
  487 = ' JOB_ID: %d'
  805 = ' Mark Height Y [mm] : %f'
  804 = ' Mark Length X [mm] : %f'
  6067 = ' Offset [m]'
  986 = ' Offset [m] : %f'
  822 = ' Print Position [m]: %f'
  823 = ' Print Stop Position [m]: %f'
  228 = ' Progress: %d %%'
  491 = ' Resolution : %d '
  192 = ' Sel PH : %d '
  13302 = ' Select header tank : %d '
  978 = ' Select headertank : %d '
  11576 = ' Selected Balance : %d '
  517 = ' Selected BL : %d '
  168 = ' Selected Group : %d '
  79 = ' Selected PC : %d '
  85 = ' Selected PG : %d '
  18812 = ' Selected PH : %d '
  8193 = ' Selected PrintModule: %d '
  215 = ' Selected Unit : %d '
  920 = ' SelHeaderTank : %d '
  2 = ' SelStorTank : %d '
  821 = ' Sensor Position [m]: %f'
  829 = ' Sensor time stamp compensation [µs]: %d'
  776 = ' Sheet detect to camera [m]: %f'
  943 = ' Sheet detect to mark [mm]: %d'
  944 = ' Sheet detect to mark [m]: %d'
  945 = ' Sheet detect to mark [m]: %f'
  826 = ' Shift start correction [m] : %f'
  827 = ' Shift start offset [m] : %f'
  13811 = ' Speed-dependent factor [s]'
  985 = ' Speed-dependent factor [s] :\n %f'
  7284 = ' Substrate thickness [m]: %f'
  819 = ' Throw Distance [mm]: %f'
  778 = ' Trigger length [sec]: %f'
  488 = ' W: %d'
  3 = ' WarningLevel'
  194 = ' X: %s [um]'
  1900 = ' X: %s [µm]'
  200 = ' Y: %s [px]'
  4807 = '! Values not persisted\n  Testing only'
  5193 = '%.1f kg'
  1205 = '%.3f kg'
  4155 = '%.4f mV/V'
  4193 = '%0.01f'
  303 = '%0.0f'
  7 = '%0.0f [%%]'
  293 = '%0.1f'
  18487 = '%0.1f [m/min]'
  7779 = '%0.1f [mbar] '
  6147 = '%0.1f [um]'
  2166 = '%0.2f'
  16761 = '%0.2f [m/s]'
  993 = '%0.3f'
  6769 = '%0.3f [m/s]'
  13150 = '%0.3f [ms]'
  1141 = '%0.4f'
  397 = '%0.6f'
  4314 = '%0.6f [ms]'
  5810 = '%0.6f [m]'
  704 = '%1.1f'
  6 = '%1.1f l'
  1138 = '%1.1f mbar'
  679 = '%1.1f mm'
  675 = '%1.1f mm/s'
  907 = '%1.1f [mbar]'
  5754 = '%1.1f [mBar]'
  39 = '%1.1f [min]'
  1038 = '%1.1f [mm]'
  1528 = '%1.1f [ms]'
  905 = '%1.1f [°C]'
  26 = '%1.2f'
  10 = '%1.2f l'
  741 = '%1.2f mm'
  917 = '%1.2f [g/cm³]'
  19 = '%1.2f [kg/l]'
  7272 = '%1.2f [m/s]'
  916 = '%1.2f [mPa*s]'
  32 = '%1.3f'
  699 = '%1.3f mm'
  913 = '%1.3f [g/cm³]'
  2489 = '%1.3f [mm]'
  915 = '%1.3f [mPa*s]'
  14861 = '%1.4f'
  735 = '%1.4f m'
  9544 = '%1.4f mm'
  12078 = '%1.4f [mm]'
  2560 = '%1.4f [m]'
  702 = '%1.6f m'
  536 = '%2.3f'
  9 = '%d'
  956 = '%D'
  6010 = '%d '
  372 = '%d %%'
  11134 = '%d [%%]'
  909 = '%d [%]'
  6448 = '%d [0.01mm]'
  1357 = '%d [0.1%%]'
  6437 = '%d [0.1mm]'
  1034 = '%d [g/m2]'
  8223 = '%d [g/m^2]'
  1035 = '%d [m/min]'
  1043 = '%d [mbar]'
  2974 = '%d [mm]'
  21 = '%d [ms]'
  7034 = '%d [m]'
  3602 = '%d [px]'
  5286 = '%d [px] '
  911 = '%d [s]'
  1059 = '%d [°C]'
  1064 = '%d [µm]'
  365 = '%d%%'
  1307 = '%ds'
  456 = '%f'
  3157 = '%f [liter]'
  10485 = '%f [m/min]'
  5388 = '%f [mm]'
  812 = '%f [m]'
  2912 = '%f [s.p.min]'
  808 = '%f [°]'
  7812 = '%f [µm/Inc]'
  14439 = '%ff'
  538 = '%i'
  27 = '%s'
  9357 = '%S'
  270 = '%s [%%]'
  319 = '%s [1..254]'
  328 = '%s [mbar] '
  322 = '%s [min]'
  612 = '%s [Min]'
  273 = '%s [ms]'
  315 = '%s [s]'
  260 = '%s%%'
  968 = '%t'
  932 = '%t%a'
  933 = '%t%b'
  353 = '%x'
  1596 = '(a refuse flow is made after a change to fill the hoses)'
  9843 = '(Hw)Enable'
  972 = '(only used if no entry found in varnish profile'
  973 = '(only used if no entry was found in varnish profile)'
  450 = '(shifted)'
  543 = '(turn off for calibration or zero scale)'
  12232 = '*'
  447 = '+'
  994 = ','
  2158 = '-'
  6598 = '-- verbos'
  19744 = '-- verbosearkDetection'
  11492 = '---'
  69 = '----'
  68 = '/'
  2302 = '0.550'
  17 = '0x%4.4x'
  9651 = '0x%4x'
  99 = '0x%x'
  441 = '1'
  6166 = '1. Activate (Drop)SpeedComp with Time set to 0\n\n2. Test1: print with production speed1\n   -> Measure displacement with Speed1\n\n3. Test2: print with production speed2\n   -> Measure displacement with Speed2\n\n4. Enter Speed and Displacement values in\n    table for Test1 and Test2\n\n5. Start new Time calculation'
  2935 = '1. Release sub menc pressure'
  495 = '1.01'
  496 = '1.05'
  497 = '1.09'
  498 = '1.13'
  499 = '1.17'
  1009 = '10'
  1010 = '12'
  1011 = '16'
  310 = '1: Vacuum pressure cannot be reached\n2: Vacuum pressure is not changing whi'
  336 = '1: Vacuum pressure cannot be reached\n2: Vacuum pressure is not changing while activation\n3: Vacuum pressure is not in defined area'
  665 = '1: Vacuum pressure cannot be reached##NEW#LINE##2: Vacuum pressure is not changing whi'
  666 = '1: Vacuum pressure cannot be reached##NEW#LINE##2: Vacuum pressure is not changing while activation##NEW#LINE##3: Vacuum pressure is not in defined area'
  440 = '2'
  1144 = '2. Deactivate level control HT'
  502 = '2.01'
  503 = '2.05'
  504 = '2.09'
  505 = '2.13'
  506 = '2.17'
  1015 = '20'
  1016 = '25'
  603 = '2nd Valve'
  74 = '2^0'
  75 = '2^1'
  451 = '3'
  9328 = '3. Purge'
  1017 = '30'
  1018 = '35'
  442 = '4'
  1145 = '4. Reactivat level and sub menc'
  3191 = '4. Reactivate level and sub menc'
  8146 = '4. Reactivate level and sub menc pos'
  12727 = '4. Reactivate level control and sub menc pos'
  1019 = '40'
  1020 = '45'
  16919 = '4p Correction Plc '
  663 = '5'
  4489 = '5. Reactivate sub menc neg'
  1021 = '50'
  1022 = '55'
  664 = '6'
  1023 = '60'
  1024 = '65'
  941 = '7'
  1025 = '70'
  1026 = '75'
  1008 = '8'
  1027 = '80'
  1028 = '85'
  1029 = '90'
  1199 = '<'
  11083 = '<-'
  448 = '='
  11216 = '>'
  444 = '>='
  9654 = '>Camera(s)'
  15769 = '>PrintPosition'
  1001 = 'A'
  722 = 'Abort'
  83 = 'Abort Transfer '
  362 = 'Acftive: %d'
  208 = 'Ack'
  3571 = 'Acknowledge'
  13067 = 'Act fill amount [cm³/min]'
  8891 = 'Act fill amount [mm³/min]'
  330 = 'Act pressure'
  661 = 'ACT VALUE CALC [°C]'
  940 = 'Act value calc [°C]'
  655 = 'ACT VALUE TEMP [0.1°C]'
  939 = 'Act value temp [0.1°C]'
  658 = 'ACT VALUE TEMP [°C]'
  577 = 'ACTIV'
  5208 = 'Activate flushing device'
  12185 = 'Activation after change'
  7529 = 'Activation after change [%]'
  2817 = 'Activation after change:'
  6604 = 'Activation delay'
  4160 = 'Activation time'
  10329 = 'Activation time supervision'
  140 = 'Active'
  1300 = 'active camera device'
  7324 = 'active camera mode'
  7209 = 'Active time'
  5594 = 'Active time after tank fill up'
  6842 = 'Active [%]'
  1036 = 'Actual job settings:'
  1039 = 'actual job settings:'
  9805 = 'Actual pulse ref'
  120 = 'Actual Pulse Reference'
  1033 = 'Actual settings:'
  8384 = 'Actual Speed'
  6725 = 'Actual speed'
  115 = 'Actual Substrate Speed'
  9679 = 'actual value [mBar]'
  110 = 'Actual Values'
  1157 = 'actual [mBar]'
  88 = 'ADD'
  89 = 'add'
  7374 = 'Add\nWhite'
  4551 = "Add PH index extension '_X'"
  12554 = 'Add vacuum pump'
  13145 = 'Add vacuum pump activation'
  2920 = 'Additional temp sensors'
  76 = 'AddWhite'
  724 = 'ADS Axis Position'
  717 = 'ADS Commands'
  0 = 'ADS InkStorage Tank'
  166 = 'ADS Mailbox VISU'
  901 = 'ADS Module Information'
  9674 = 'ADS PG shift'
  2259 = 'ADS PU shift'
  723 = 'ADS Settings'
  9294 = 'Aerosol measurement'
  651 = 'after purge'
  1058 = 'Air temperature setting'
  117 = 'Alignments'
  6201 = 'All enabled CBs are in OP'
  892 = 'All Module OK'
  19755 = 'ALL Persistent Values!!!!'
  890 = 'AMS NetId'
  5680 = 'AnalogMaxDigit'
  4820 = 'arw'
  2081 = 'AS'
  262 = 'Auto'
  574 = 'AUTO'
  1046 = 'auto'
  381 = 'Auto dest. path'
  382 = 'Auto destination path'
  593 = 'AUTO EXCHANGE'
  671 = 'AUTO/MANU CONTROL'
  718 = 'Automatic Mode'
  2606 = 'AutomaticMode or ManualTeach'
  11632 = 'AutomaticMode or ManualTeach or SimEnable'
  860 = 'Auxiliary Encoder'
  798 = 'Average Angle'
  52 = 'B'
  17116 = 'Back'
  14 = 'Balance'
  2271 = 'BALANCE'
  247 = 'Balance\nVISU_BALANCE'
  559 = 'Balance 1'
  560 = 'Balance 2'
  10235 = 'Balance : %s'
  30 = 'Balance Configuration'
  512 = 'Balance Error'
  508 = 'Balance OK'
  509 = 'Balance Warning'
  1769 = 'Barcode scanned label ID'
  1764 = 'Barcode scanned string'
  1766 = 'Barcode scanned tank index'
  1761 = 'Barcode scanner receive data: %d'
  565 = 'Beckhoff terminal WcState error'
  13353 = 'bInvertedX'
  514 = 'Bit 0: 16#01: -\nBit 1: 16#02: No level after maintenance\nBit 2: 16#04: Headertank empty\nBit 3: 16#08: Headertank low\nBit 4: 16#10: Storage tank warning level\nBit 5: 16#20: Storage tank error level\nBit 6: 16#40: Storage tank missing\nBit 7: 16#80: -'
  525 = 'Bit 0: 16#01: -\nBit 1: 16#02: Send data error\nBit 2: 16#04: Receive no data\nBit 3: 16#08: Balance in motion\nBit 4: 16#10: Balance not connected\nBit 5: 16#20: Buffer full\nBit 6: 16#40: Framin fault\nBit 7: 16#80: Over run error'
  73 = 'Bit per Pixel'
  5263 = 'bI_CANopen_CleaningStart'
  12638 = 'bI_CANopen_EnablingOn'
  1100 = 'bI_CANopen_Engaged'
  1102 = 'bI_CANopen_EStop'
  1104 = 'bI_CANopen_MessageReset'
  1105 = 'bI_CANopen_PinningClosed'
  1101 = 'bI_CANopen_PrintEnabled'
  15388 = 'bI_CANopen_PrintEnablIbEAP_PrintEIbEAP_PrintEnabled M2'
  1099 = 'bI_CANopen_ShutDownActive'
  1103 = 'bI_CANopen_StandbyActive'
  6499 = 'bI_EStopOk'
  6476 = 'bI_MachineReady'
  6504 = 'bI_ReleasePurge'
  6470 = 'bI_RunningMode'
  6482 = 'bI_SafetyCover_CU'
  6487 = 'bI_SafetyCover_Inlet'
  6493 = 'bI_SafetyCover_Outlet'
  6510 = 'bI_SheetCameraTeach'
  6516 = 'bI_StopPrinter'
  463 = 'BlockBase:'
  462 = 'BlockTypes:'
  774 = 'bL_CameraNewResult'
  2543 = 'bL_ProductionMode'
  6246 = 'bL_ZAxisPosOverridePurge'
  146 = 'Board enable'
  902 = 'Boundary Errors: %d'
  5277 = 'bO_CANopen_CleaningActive'
  5272 = 'bO_CANopen_CleaningAllowed'
  1111 = 'bO_CANopen_EngagingAllowed'
  1114 = 'bO_CANopen_PrintPosition'
  1112 = 'bO_CANopen_ShutdownReady'
  1113 = 'bO_CANopen_StandbyReady'
  8260 = 'bO_CU_Referenced'
  179 = 'bO_PauseCanEx'
  184 = 'bO_PauseExec'
  8238 = 'bO_PrinterReady'
  8267 = 'bO_Sleep'
  177 = 'bO_StartCanEx'
  182 = 'bO_StartExec'
  178 = 'bO_StopCanEx'
  183 = 'bO_StopExec'
  8253 = 'bO_VaccumPumpON'
  8245 = 'bO_WasteSheet'
  8083 = 'BS'
  210 = 'Busy'
  375 = 'busy'
  13078 = 'by calc'
  19400 = 'by calculation'
  411 = 'c'
  6619 = 'C'
  744 = 'C1'
  743 = 'C2'
  710 = 'Ca/Pu'
  18477 = 'Calculate new time'
  1431 = 'Calculate new Time'
  13966 = 'calculated by Cyclinder'
  7985 = 'calculated by cyclinder'
  33 = 'Calibration'
  518 = 'Calibration Scale'
  5997 = 'Calmar update'
  12287 = 'Cam device: %s'
  2799 = 'Cam mode: %s'
  15228 = 'Cam Simulation'
  1190 = 'Cam valid'
  5849 = 'CamDone LastMark'
  11355 = 'Camera'
  779 = 'Camera BS - AS'
  7188 = 'Camera selection'
  19366 = 'Cameras'
  11139 = 'CameraToPrintUnit'
  2957 = 'CameraTrigger'
  16237 = 'CameraTrigger active'
  5607 = 'CamToPU'
  921 = 'CanEx'
  1110 = 'CANopen Interface CALMAR <-> MACHINE'
  1126 = 'CANopen_NodeState'
  922 = 'CanStop'
  9349 = 'Capping position'
  965 = 'Capping postion'
  707 = 'CappPurge Position'
  544 = 'case sensitive'
  71 = 'CB'
  572 = 'CH VALVE CLEANER'
  573 = 'CH VALVE CONTROL AIR'
  527 = 'Ch1'
  528 = 'Ch2'
  529 = 'Ch3'
  530 = 'Ch4'
  531 = 'Ch5'
  532 = 'Ch6'
  533 = 'Ch7'
  534 = 'Ch8'
  929 = 'Change'
  934 = 'Change Printline1'
  1004 = 'Change Printline1&2'
  935 = 'Change Printline2'
  199 = 'Channel'
  34 = 'Channel Configuration'
  539 = 'Channel ID'
  5449 = 'Charged Columns'
  8294 = 'Check delay'
  6636 = 'CheckDelay'
  261 = 'Circl'
  281 = 'Circulation'
  320 = 'cI_PurgeRepeats'
  708 = 'Clean'
  697 = 'Clean Active'
  719 = 'Clean after Capping'
  720 = 'Clean after Purge'
  684 = 'Clean Head'
  5415 = 'Clean head'
  254 = 'Clean Head\nVISU_CH'
  8522 = 'Clean head (max %d)'
  725 = 'Clean Row 1'
  726 = 'Clean Row 2'
  11428 = 'Clean sequence'
  683 = 'Clean Shiny'
  711 = 'Clean Unit'
  253 = 'Clean Unit\nVISU_CU'
  15882 = 'Clean unit (max %d)'
  698 = 'Clean Wanne'
  14428 = 'CleanCappPosition'
  259 = 'Cleaner'
  567 = 'CLEANER'
  7450 = 'Cleaner air bubble detection'
  8549 = 'Cleaner CommandCanEx'
  977 = 'Cleaner fill'
  629 = 'CLEANER PUMP'
  4468 = 'Cleaner pump'
  570 = 'Cleaner-'
  11419 = 'CleanHead'
  747 = 'Cleaning'
  583 = 'CLEANING  %'
  10965 = 'Cleaning capping pos.'
  2402 = 'CLEANING CLEANER PUMP'
  694 = 'Cleaning Operations'
  740 = 'Cleaning Safe '
  5877 = 'Cleaning tub'
  10350 = 'Cleaning tub (max %d)'
  706 = 'CleanPosition 2'
  705 = 'CleanPosition1'
  11400 = 'CleanUnit'
  81 = 'Cmd : 0x%8.8x'
  93 = 'Cmd_Data'
  94 = 'Cmd_Fire'
  7325 = 'Code: %d'
  207 = 'COE COMMAND'
  209 = 'COE FLAGS'
  357 = 'CoE Service'
  342 = 'CoeAdr'
  344 = 'CoeLength'
  343 = 'CoeSubAdr'
  352 = 'CoeValue'
  966 = 'Color ID'
  1396 = 'Column Precharge'
  390 = 'Com'
  5379 = 'COM BALANCE'
  4156 = 'Com state'
  523 = 'COMM Balance'
  248 = 'COMM Balance\nVISU_COMM_BALANCE'
  1908 = 'Command'
  163 = 'COMMANDS'
  132 = 'COMMANDS (overwritten)'
  391 = 'Communication error'
  1052 = 'Compressor setpoint %1.1f [V]'
  4895 = 'Conditions'
  4044 = 'Conditions:'
  8489 = 'Configuration'
  7795 = 'Confirm empty HT'
  9558 = 'constant'
  569 = 'container'
  306 = 'Contr operative'
  485 = 'Controller'
  370 = 'Controller Board enabled'
  947 = 'Conversion'
  903 = 'Conversion Errors: %d'
  510 = 'CONVERSIONS'
  807 = 'Conveyor Speed'
  878 = 'Conveyor Speed Pg1'
  868 = 'Conveyor Speed [m/s]: %f'
  866 = 'corr : %0.6f'
  591 = 'Correct headertank must be\nconnected manually'
  25 = 'Correction Factor'
  11413 = 'Correction [mbar]'
  1135 = 'CorrectionFactor'
  11397 = 'Counter'
  8478 = 'ct'
  3579 = 'CT'
  7237 = 'CT @Deformation (more corrections follow @Print!)'
  8221 = 'CT @Deformation (more corrections followed @Print!)'
  8596 = 'CT create'
  3207 = 'CT Create'
  12836 = 'CT destroy'
  3546 = 'CT Destroy'
  1850 = 'CT PrintRef'
  4803 = 'ctrl err'
  785 = 'Current Angle'
  8940 = 'Current Column Pos'
  10240 = 'Current CT'
  10438 = 'Current position'
  5063 = 'Current step'
  786 = 'Current Y Shift'
  1572 = 'Cycle'
  6944 = 'cycle pos x'
  389 = 'D'
  13198 = 'd=%f'
  14919 = 'Date & Time'
  621 = 'DE-AIR'
  622 = 'DE-AIR TIME'
  623 = 'DE-AIR WAIT TIME'
  2419 = 'Dead/Add Time'
  4013 = 'Dead/Add Time [ms]'
  11659 = 'Debug'
  21105 = 'Debug & Simulation'
  761 = 'Debug counter index found: %d'
  762 = 'Debug counter index not found: %d'
  961 = 'Debug FIFO Cam1 PG1 (level: %d)'
  962 = 'Debug FIFO Cam2 PG1 (level: %d)'
  775 = 'Debug FIFO PG1 (level: %d)'
  942 = 'Debug FIFO PG2 (level: %d)'
  16219 = 'Debug mode: %s'
  5718 = 'Def fill amount [mm³/min]'
  239 = 'Default file'
  3703 = 'Default fill amount [mm³/min]'
  1152 = 'Default HT temp'
  4210 = 'Default HT temp [1/10 °C]'
  5777 = 'Default pump speed'
  2602 = 'Default pump speed [digit]'
  11934 = 'Default sub men neg'
  9276 = 'Default sub men neg [1/10 mbar'
  1155 = 'Default sub men neg [1/10 mbar]'
  11642 = 'Default sub menc pos'
  6724 = 'Default sub menc pos [1/10 mbar]'
  231 = 'Define PH mask files'
  245 = 'Degassing / Meniscus\nVISU_VACUUM'
  277 = 'Delay'
  5312 = 'Delay BiBchange'
  2752 = 'Delay flow heater'
  1320 = 'Delay lock cleaning'
  82 = 'Delete Current Job'
  4766 = 'Delta'
  17633 = 'Delta mark 1 to 2 [SubPx]'
  1129 = 'Delta Mark-Print'
  701 = 'Delta P'
  880 = 'Delta Position'
  885 = 'Delta Position max.'
  884 = 'Delta Position min.'
  992 = 'DeltaX angle'
  991 = 'DeltaX [mm]'
  1075 = 'DEM engaged'
  1080 = 'DEM not engaged (Service)'
  10191 = 'Desc'
  50 = 'Desired Copies : %d'
  211 = 'Dest'
  373 = 'Dest.'
  3463 = 'DestFilePath'
  219 = 'Destination'
  379 = 'Destination path'
  5100 = 'Detail Views'
  16410 = 'detected'
  7234 = 'detected marks'
  12392 = 'DetectToCam'
  11747 = 'DetectToCamera'
  54 = 'Device Address : %d'
  12363 = 'DevOpActive'
  648 = 'Dgas'
  563 = 'Dgas pressure OK'
  296 = 'Dgas valve'
  1139 = 'Disable'
  1185 = 'Disable delay module3'
  11190 = 'Disable DriftControl'
  1171 = 'Disable left SLM'
  2820 = 'disable ModuleSynchronisation'
  2726 = 'Disable ModuleSynchronisation'
  11545 = 'Disable ModuleSynchronisation (start, stop)'
  6432 = 'Disable right SLM'
  10093 = 'Disable trigger M3'
  9310 = 'Disable trigger modele3'
  16750 = 'Disable trigger module3'
  2162 = 'Displacement'
  12778 = 'Distance mark 1 to 2 [mm]'
  748 = 'distance to Print Unit'
  669 = 'DO'
  749 = 'Dog-ear detection: enable'
  152 = 'Done'
  482 = 'Download'
  367 = 'Download Busy'
  368 = 'Download Error'
  366 = 'Download progress'
  403 = 'dp\n---\ndt'
  10270 = 'Drift control'
  9832 = 'Drive time: %s'
  817 = 'Drop Speed Comp'
  64 = 'DropSize : %d'
  4615 = 'DropSpeed'
  13254 = 'DropSpeed Compensation'
  12555 = 'DropSpeed Compensation [m/s]/[ms]'
  1196 = 'DropSpeed Setup'
  4971 = 'DropSpeed [m/s]'
  14399 = 'DropSpeedCorr'
  15240 = 'DropSpeedCorrection'
  3206 = 'DropSpeedCorrection [m/s] []'
  2684 = 'DropSpeedCorrection [m/s]/[ms]'
  63 = 'Dummy'
  2828 = 'Duration mark 1 to 2'
  16577 = 'Duration mark 1 to 2 [ms]'
  3002 = 'Duration mark 1 to 2 [s]'
  783 = 'DVT Sheet Rotation'
  4842 = 'dX shift (points)'
  7303 = 'dx: %0.3f'
  1197 = 'dx:%0.3f'
  12149 = 'dx=%0.4f'
  5761 = 'dx=%0.5f'
  14558 = 'dx=%d'
  16207 = 'dx=%f'
  14629 = 'dy: %0.3f'
  10064 = 'dy:%0.3f'
  14821 = 'dy=%0.4f'
  15313 = 'dy=%0.5f'
  7404 = 'dy=%f'
  53 = 'E'
  18481 = 'e state'
  1176 = 'EAP Interface CALMAR <-> MACHINE'
  824 = 'Eject'
  825 = 'Eject All'
  799 = 'Eject angle range error'
  8405 = 'EL5101 simulation'
  685 = 'EL7201'
  360 = 'Elems'
  361 = 'Elems: %d'
  9770 = 'Emergency Stop'
  6261 = 'EmergencyStop active'
  926 = 'Empty'
  8 = 'Enable'
  142 = 'ENABLE'
  28 = 'Enable Balance Link'
  4131 = 'Enable barcode scanner'
  2655 = 'Enable blue'
  2501 = 'Enable Correction'
  266 = 'Enable Dgas valve'
  3450 = 'Enable donwloader'
  123 = 'Enable Filter'
  4043 = 'Enable green'
  800 = 'Enable HW Mode'
  294 = 'Enable ink pump'
  545 = 'Enable Main Dgas Valve'
  96 = 'Enable Manual Data'
  97 = 'Enable Manual Pulse'
  9074 = 'Enable Motion Simulation'
  8043 = 'Enable orange'
  193 = 'Enable PH'
  313 = 'Enable purge'
  605 = 'ENABLE PURGE'
  268 = 'Enable ramp'
  2016 = 'Enable red'
  408 = 'Enable simulation'
  8850 = 'Enable Testing'
  236 = 'Enable updater'
  102 = 'Enable Vaccum Pump'
  234 = 'Enabled'
  7765 = 'Enabled compensation'
  1070 = 'Enabling settings'
  1003 = 'Enabling System'
  9778 = 'EnAutoStartPrinting'
  395 = 'Enc.Res.[p/um]'
  12315 = 'Encoder (radius, resolution, )'
  8505 = 'Encoder Compensation'
  113 = 'Encoder Resolution'
  14488 = 'Encoder speed compensation factor'
  5880 = 'Encoder speed compensation reference speed'
  859 = 'Encoder Wheel'
  11490 = 'Encoder wheel diameter'
  398 = 'Encoder-'
  14442 = 'EncoderCyilinderDiameter [mm]'
  7997 = 'EncoderCylinderDiameter [mm]'
  9966 = 'EncoderResolution'
  2234 = 'EncoderResolution  [µm/Inc]'
  11113 = 'EncoderResolution [µm/Inc]'
  13259 = 'EncRes %f'
  1636 = 'EncSpeedCorrection'
  417 = 'Endless'
  5930 = 'Engaged'
  7298 = 'EnOnly'
  714 = 'Enter Capping'
  4621 = 'Err: %d'
  7584 = 'ErrId: %d'
  40 = 'Error'
  376 = 'error'
  5258 = 'Error active'
  7548 = 'Error Code'
  1158 = 'Error level'
  5510 = 'Error Message active'
  465 = 'Error:'
  358 = 'ErrorCode'
  731 = 'EStop'
  689 = 'EStop Ok'
  59 = 'ETH'
  891 = 'EtherCAT Configuration'
  590 = 'EXCHANGE'
  521 = 'Exchange Type'
  923 = 'Exec'
  2082 = 'Execute device reset only in CU park position!'
  6374 = 'Execute device reset only in exit capping!'
  14686 = 'Execute device reset only in PU service position!'
  928 = 'Execute flush'
  16510 = 'Execute purge'
  18335 = 'Exeeds max. speed=%f'
  12796 = 'Exhaust'
  11482 = 'Exhaust active'
  10280 = 'Exhaust FU error'
  1734 = 'Exhaust system'
  6652 = 'Exhaust system module 1'
  15247 = 'Exhaust system module 2'
  1156 = 'Exhaust vacuum measurement'
  2867 = 'Exhaust vacuum measurement 0-50mBar'
  3763 = 'Exhaust vacuum warn/error'
  715 = 'Exit Capping'
  72 = 'F'
  638 = 'factor'
  524 = 'Fault Ack.'
  513 = 'Fault Acknowledge'
  4816 = 'fb err'
  6768 = 'FB_PositionMaster'
  754 = 'fb_SegmentSlave[PG1].Index'
  757 = 'fb_SegmentSlave[PG2].Index'
  10135 = 'FB_Worker'
  36 = 'Feedback'
  4662 = 'feedback [mBar]'
  15781 = 'fHeight'
  974 = 'Fil ink'
  975 = 'Fil varnish'
  238 = 'File per PH'
  383 = 'File per printhead'
  265 = 'Fill'
  581 = 'FILL %'
  11658 = 'Fill amount history [mm³/min]'
  2763 = 'Fill amount [cm³/min]'
  4465 = 'Fill amount [mm³/min]'
  979 = 'Fill cleaner'
  1925 = 'Fill headertank'
  558 = 'FILL VARNISH'
  976 = 'Fill varnish'
  15193 = 'Fill varnish activated'
  636 = 'FILL VARNISH PUMP'
  3783 = 'Filter supervision'
  5240 = 'Filter supervision BiB / RT'
  10977 = 'Filter supervision BiB => RT'
  1660 = 'Filter supervision RT => HT'
  134 = 'FLAGS'
  10347 = 'Flash orange'
  16158 = 'fLength'
  1069 = 'Flow monitor delay'
  1068 = 'Flow monitor delay [ms]'
  927 = 'Flush'
  332 = 'Flush (through ph)'
  333 = 'Flush time'
  2772 = 'FlushingState'
  58 = 'FoE'
  422 = 'Foe'
  212 = 'FOE COMMAND'
  213 = 'FOE FLAGS'
  586 = 'For auto select tank'
  730 = 'Force Close'
  14353 = 'Force HwReady'
  729 = 'Force Open'
  1134 = 'Format Length'
  1691 = 'FormatLength'
  4688 = 'FormatTrigger'
  222 = 'FPGA Update'
  11995 = 'fPosX'
  4329 = 'fPosY'
  12999 = 'fPrintStartOffset'
  8188 = 'fPrintXOffsetMachine'
  6987 = 'free'
  226 = 'From PC:'
  7569 = 'FSM State PC[%d]'
  220 = 'FW Update'
  1178 = 'Gap'
  108 = 'General Settings'
  1148 = 'GeneralShiftX'
  13867 = 'GeneralShiftX [µm]'
  6168 = 'GeneralShiftY'
  14591 = 'GeneralShiftY [µm]'
  519 = 'Get weight'
  535 = 'Get Weight'
  421 = 'Gigabit'
  8756 = 'Global Settings'
  7612 = 'Global status'
  4206 = 'Gross Weight:'
  84 = 'Group Cmd'
  494 = 'Group MODE'
  857 = 'Group1'
  858 = 'Group2'
  17119 = 'GroupBox'
  7927 = 'h: %0.3f'
  5110 = 'h:%0.3f'
  15957 = 'h=%0.4f'
  171 = 'HARDWARE'
  5131 = 'Hardware'
  406 = 'Hardware Encoder input'
  6909 = 'Head'
  3904 = 'Head base plate gap to roller table [m]: %f'
  4341 = 'Head base plate to roller table'
  14853 = 'Head base plate to roller table [mm]'
  10221 = 'Head base plate to roller table [m]'
  16374 = 'Head base plate to table gap [mm]'
  4730 = 'Head base plate to table [mm]'
  3625 = 'Head Gap [mm]'
  13438 = 'Head Offset Plate [mm]'
  5194 = 'Head Offset Plate [m]'
  2652 = 'Head offset to base plate [m]: %f'
  3353 = 'Head set counter value: %d'
  10161 = 'HEADERTANK'
  546 = 'Headertank 1'
  548 = 'Headertank 2'
  550 = 'Headertank 3'
  552 = 'Headertank 4'
  554 = 'Headertank 5'
  556 = 'Headertank 6'
  760 = 'Heartbeat'
  161 = 'Heater enable'
  653 = 'HEATING'
  938 = 'Heating'
  244 = 'Heating\nVISU_TEMPERATUR'
  652 = 'HEATING HEADERTANK'
  969 = 'Heating ON time'
  971 = 'Heating ON time [ms]'
  967 = 'Heating period'
  970 = 'Heating period [ms]'
  656 = 'HEATING PRINT HEAD PLATE'
  1057 = 'Height setting'
  7555 = 'HIB Remote Update'
  6007 = 'HIB update'
  642 = 'histeresis [0,1°C]'
  1153 = 'History'
  1150 = 'HT area [mm²]'
  3255 = 'HT back level'
  1146 = 'HT back long [°C]'
  6159 = 'HT back short [°C]'
  5094 = 'HT front long [°C]'
  10231 = 'HT front short [°C]'
  10248 = 'HT passing [°C]'
  2587 = 'HT refuse'
  11818 = 'HT surface [mm²]'
  10219 = 'HT temp'
  9841 = 'HT test amount [cm³/min]'
  2496 = 'HT test amount [mm³/min]'
  405 = 'HW'
  125 = 'HW Encoder'
  2960 = 'HwEnable'
  12780 = 'HwReady'
  8700 = 'Hysteresis [mbar]'
  388 = 'I'
  1132 = 'I-Gain'
  11288 = 'IbEAP_CleaningStart M2'
  15820 = 'IbEAP_CleaningStart M3'
  10115 = 'IbEAP_Engage M2'
  9437 = 'IbEAP_Engage M3'
  4235 = 'IbEAP_Engaged'
  9617 = 'IbEAP_Engaged M2'
  10431 = 'IbEAP_Engaged M23'
  7259 = 'IbEAP_Engaged M3'
  5659 = 'IbEAP_EStop'
  4716 = 'IbEAP_MessageReset'
  11953 = 'IbEAP_PinningClosed M2'
  14012 = 'IbEAP_PinningClosed M3'
  7162 = 'IbEAP_PrintEnable M2'
  16427 = 'IbEAP_PrintEnable M3'
  15661 = 'IbEAP_PrintEnabled M2'
  2964 = 'IbEAP_PrintEnabled M3'
  5588 = 'IbEAP_PrintMarksExist M2'
  8618 = 'IbEAP_PrintMarksExist M3'
  9463 = 'IbEAP_ShutDownActive'
  16498 = 'IbEAP_SpliceDetected M2'
  13908 = 'IbEAP_SpliceDetected M3'
  8509 = 'IbEAP_StandbyActive'
  8826 = 'IbEAP_TargetSpeedReached'
  10276 = 'IbEStop'
  7563 = 'IbMachineActive'
  14174 = 'IbMessageReset'
  6426 = 'IbPhEnableBlack'
  1165 = 'IbPhEnableCyan'
  1513 = 'IbPhEnableMagenta'
  9734 = 'IbPhEnableWhite'
  10218 = 'IbPhEnableYellow'
  9071 = 'IbPurgeAllowed'
  7629 = 'IbPurgeCommand'
  3742 = 'IbPurgeEnableBlack'
  14251 = 'IbPurgeEnableCyan'
  14811 = 'IbPurgeEnableMagenta'
  10094 = 'IbPurgeEnableWhite'
  1167 = 'IbPurgeEnableYellow'
  9262 = 'IbStartPosition'
  18013 = 'Id'
  147 = 'Idle'
  13165 = 'Idx'
  424 = 'Image Depth'
  425 = 'Image Width'
  48 = 'ImageDepth : %d'
  49 = 'ImageWidth : %d'
  156 = 'Img-Offset'
  1183 = 'ImgLength'
  15455 = 'Impl.'
  733 = 'In     Out'
  21992 = 'In jet print system CALMAR'
  6859 = 'InArea'
  204 = 'Index'
  13591 = 'InEAP_FormatLength'
  1475 = 'InEAP_FormatLength: %0.4f [m]'
  2005 = 'InEAP_LateralRegister'
  10767 = 'InEAP_Module2ToModule3'
  6222 = 'InEAP_NeutralFibreFactor'
  4588 = 'InEAP_OperatingMode'
  12393 = 'InEAP_SubstrateThickness'
  11615 = 'InEAP_SubstrateWidth'
  3434 = 'InEAP_TargetSpeed'
  3556 = 'InEAP_WatchdogCycleIndex'
  6925 = 'InEAP_WebStretchFactor'
  657 = 'INFEED'
  660 = 'INFEET'
  56 = 'Infinite'
  889 = 'Inhib Sensor1'
  879 = 'Inhib Sensor2'
  871 = 'InhibAct [ms]: %d'
  1262 = 'Inhibit trigger'
  869 = 'InhibTime [ms]: %d'
  4321 = 'Init'
  15016 = 'Init ok'
  4150 = 'Init test'
  457 = 'InitOK'
  2261 = 'INK'
  9965 = 'Ink'
  279 = 'Ink\npump'
  1637 = 'Ink circulation'
  11768 = 'INK CMYK'
  13 = 'Ink Color ID'
  20 = 'Ink Density'
  4538 = 'Ink jet print system CALMAR'
  4734 = 'INK W'
  3063 = 'INK White'
  816 = 'InkSys Ready'
  255 = 'InkSystem'
  1066 = 'Inlet'
  13124 = 'InPassNumber'
  3500 = 'Input Resolution'
  1149 = 'Input test'
  1115 = 'Inputs'
  1902 = 'Inspection System'
  363 = 'Inst: %d'
  693 = 'Interlock'
  4159 = 'inverted'
  6150 = 'inverted X'
  1195 = 'invertedx'
  750 = 'IP address'
  11599 = 'ix'
  4790 = 'J'
  386 = 'Job'
  46 = 'Job ID : %d'
  490 = 'Job List'
  387 = 'Job loaded'
  6151 = 'Job Loading: %s'
  483 = 'Job Status'
  3573 = 'JobActive'
  423 = 'JobId'
  432 = 'JobLength'
  4454 = 'JobLoaded'
  6002 = 'JobManagement'
  216 = 'JobShiftX'
  217 = 'JobShiftY'
  10484 = 'JobStart (manual trig)'
  5963 = 'JobStop (manual trig)'
  11398 = 'Key'
  7660 = 'Ki time'
  19077 = 'l=%0.4f'
  4340 = 'Label scan needed'
  10125 = 'LateralRegister'
  2351 = 'LED base timer (muitple of 2ms)'
  206 = 'Length'
  3520 = 'Length check'
  6260 = 'Length in Job'
  4463 = 'Length in Machine'
  13708 = 'Length Missmatch'
  4787 = 'Length [subpix]: %3.2f'
  765 = 'Length: %d [ms]'
  4310 = 'Level under set point [mm]'
  6296 = 'Level under setpoint [mm]'
  737 = 'LimitDN'
  736 = 'LimitUP'
  17634 = 'Link'
  5281 = 'lI_CANopen_FormatLength '
  1106 = 'lI_CANopen_LateralRegister'
  1107 = 'lI_CANopen_SubstrateThickness'
  1108 = 'lI_CANopen_SubstrateWidth'
  1109 = 'lI_CANopen_WebStretchFactor'
  5109 = 'lI_ImageDepth'
  5300 = 'lL_ImageDepthPx from PUC'
  5295 = 'lL_SubstrateLenPx from CANopen'
  17382 = 'lL_ToleranceLenPx'
  470 = 'LOAD'
  2972 = 'Log time intervall'
  18927 = 'Logger'
  11756 = 'LogLevel'
  5764 = 'LogLevel: %s'
  8854 = 'Low intense mode'
  1118 = 'lO_CANopen_MaxWebSpeed'
  1117 = 'lO_CANopen_VarnishQuantity'
  8103 = 'lsq=%0.4f'
  17552 = 'ltr=%0.4f'
  6995 = 'lx=%0.4f'
  13612 = 'ly=%0.4f'
  290 = 'M'
  180 = 'm/s: %0.2f'
  16061 = 'M2: Pinning closed'
  3879 = 'M3: Pinning closed'
  256 = 'Machine'
  15026 = 'MAchine'
  1030 = 'machine\nspeed\n[m/min]'
  6479 = 'Machine Interface'
  1231 = 'Machine Print Overview'
  12211 = 'Machine Ready'
  3025 = 'Machine Sim'
  4332 = 'Machine Sim '
  9707 = 'Machine Sim %d'
  16705 = 'Machine Sim OK '
  10239 = 'Machine Sim Radom'
  13712 = 'Machine started'
  20139 = 'MachineComm'
  3709 = 'MachineComm Sim'
  1179 = 'MachineStopped'
  14491 = 'Main'
  299 = 'Main controller %s'
  427 = 'Maint.Images'
  15 = 'Maintenance'
  1137 = 'Maintenance Meniscus'
  22 = 'Maintenance Timeout'
  267 = 'Manu'
  579 = 'MANU'
  6402 = 'MANU CONTROL'
  1045 = 'manual'
  1002 = 'Manual move'
  8502 = 'Manual Start PM1'
  15154 = 'Manual Start PM2'
  14480 = 'Manual Teach'
  5389 = 'Manual Teach Trigger'
  758 = 'Manual Trigger: (response time %s )'
  12902 = 'Manually activtaion'
  464 = 'Mapping Generator'
  893 = 'Mapping Overflow'
  1290 = 'Mark bits'
  795 = 'Mark Detection'
  984 = 'Mark detection'
  1187 = 'Mark orientation'
  8258 = 'Mark sensors'
  16062 = 'MarkCamera'
  8898 = 'MarkDefinition'
  17557 = 'MarkDefinition '
  1627 = 'MarkDefinition Entries'
  20000 = 'MarkDetection'
  6617 = 'MarkLength [mm]: %3.2f'
  15941 = 'Marks Inverted'
  10171 = 'Marks to adjust : %d'
  11321 = 'Marks to stop: %d'
  9087 = 'marks valid'
  11470 = 'MarkState'
  197 = 'Mask File'
  981 = 'Mask file'
  232 = 'Mask Update'
  7504 = 'Master module idx'
  116 = 'Master Position'
  9579 = 'Master position'
  14368 = 'Master position [SubPx]:: %d'
  10569 = 'Master position [µm]:: %1.1f'
  4786 = 'MasterModule'
  272 = 'Max'
  626 = 'Max %'
  633 = 'Max digit'
  9524 = 'Max numbers of logs'
  329 = 'Max pressure'
  646 = 'Max volt'
  791 = 'Max Y Shift'
  3075 = 'Max. Speed is: %s'
  18832 = 'Max. Speed m/s'
  13601 = 'Max. Speed [m/s]'
  12274 = 'max: %d'
  14892 = 'Measurement'
  784 = 'Memory Offset'
  650 = 'Menc main'
  4525 = 'Menc neg'
  6435 = 'Menc pos'
  2118 = 'MencShutOffValve force FALSE'
  7743 = 'MencShutOffValve force TRUE'
  271 = 'Min'
  625 = 'Min %'
  632 = 'Min digit'
  327 = 'Min pressure'
  645 = 'Min volt'
  10496 = 'Min. Speed for Production'
  11339 = 'Min. Speed for Production [m/min]'
  7865 = 'Min. speed production [m/min]'
  1193 = 'Missed'
  35 = 'Mixer'
  37 = 'Mixer on time'
  38 = 'Mixer wait time'
  98 = 'Mode configuration'
  314 = 'Mode Manu'
  606 = 'MODE MANU'
  8621 = 'Modul 2'
  12678 = 'Modul 3'
  11758 = 'Module %d'
  1191 = 'Module %s'
  14156 = 'Module 1 (2)'
  12260 = 'Module 2'
  12265 = 'Module 2 ()'
  9306 = 'Module 2 (3)'
  9555 = 'Module 3'
  16997 = 'Module Base'
  19210 = 'Module Details'
  894 = 'Module Handler'
  460 = 'Module ident. number'
  22051 = 'Module Master (Job and Production)'
  8247 = 'Module position\n- Alignments (display)\n- Setting (y-Shift of Module)\n- '
  1186 = 'Module to module adjust [µm]'
  13999 = 'Module to module Y adjust [SubPx]'
  13151 = 'Module to module Y adjust [µm]'
  10097 = 'Module WEU'
  19574 = 'Module=%d'
  5856 = 'Modules'
  341 = 'Monitoring of pump activation'
  686 = 'MOTION'
  7218 = 'Motion'
  17228 = 'Motion specific\n- Axis (diamater, resolution, enc comp.)'
  540 = 'MotionCount  '
  691 = 'Move Done'
  673 = 'MoveEnable'
  135 = 'Moving'
  522 = 'MUX ID'
  70 = 'N'
  196 = 'Name of mask file in folder\n05_Mask with extension  .msk'
  459 = 'Name:'
  900 = 'Nbr Mappings'
  899 = 'Nbr Modules'
  467 = 'Nbr:'
  541 = 'NC_Count  '
  5268 = 'Net Weight:'
  9250 = 'Neutral fibre supervision'
  1194 = 'NeutralFiber'
  9686 = 'NeutralFiberFactor [%]'
  17046 = 'nId'
  696 = 'No Liquid'
  9545 = 'NoCamera'
  22010 = 'None'
  13171 = 'normal'
  3138 = 'not engaged (Service)'
  420 = 'Nothing'
  16262 = 'Number of modules'
  7300 = 'O'
  7240 = 'ObEAP_CleaningActive M2'
  13228 = 'ObEAP_CleaningActive M3'
  16642 = 'ObEAP_CleaningAllowed M2'
  14932 = 'ObEAP_CleaningAllowed M3'
  15304 = 'ObEAP_EngagingActive M2'
  7926 = 'ObEAP_EngagingActive M3'
  7601 = 'ObEAP_EngagingAllowed M2'
  8194 = 'ObEAP_EngagingAllowed M3'
  5471 = 'ObEAP_ErrorActive'
  15972 = 'ObEAP_EStop'
  2833 = 'ObEAP_PrintPosition M2'
  5491 = 'ObEAP_PrintPosition M3'
  1177 = 'ObEAP_PrintReady M2'
  5250 = 'ObEAP_PrintReady M3'
  16120 = 'ObEAP_ShutdownReady'
  12649 = 'ObEAP_StandbyReady'
  8986 = 'ObEAP_WarnungActive'
  7339 = 'ObErrorMsgActive'
  3436 = 'ObPrinterJobLoaded'
  2428 = 'ObPrinterPrinting'
  7942 = 'ObPrinterReady'
  10769 = 'ObPrintReady'
  8375 = 'ObPurgeActive'
  6496 = 'ObWarningMsgActive'
  413 = 'of'
  4393 = 'Off delay'
  153 = 'OFFSET'
  195 = 'Offset'
  44 = 'Offset Address : %d'
  1164 = 'OfImageLengthJob'
  7013 = 'OfYOffsetPass'
  7421 = 'OnEAP_MasterSpeed M2'
  12229 = 'OnEAP_MasterSpeed M3'
  7974 = 'OnEAP_MaxWebSpeed'
  11987 = 'OnEAP_OperatingMode'
  11795 = 'OnEAP_PrintMarkPosBits M2'
  8809 = 'OnEAP_PrintMarkPosBits M3'
  12676 = 'OnEAP_VarnishQuantity M2'
  1466 = 'OnEAP_VarnishQuantity M3'
  7305 = 'Only enabled PCs'
  14046 = 'OnNumberPassJob'
  732 = 'Open Shutter'
  1044 = 'operating mode'
  1050 = 'Operating mode'
  716 = 'Operation'
  511 = 'OPERATIONS'
  946 = 'Operations'
  1078 = 'Option'
  1079 = 'Option / not existing'
  8015 = 'Orange: LED green activation [%]'
  5120 = 'Orange: LED red activation [%]'
  659 = 'OUTLET'
  1067 = 'Outlet'
  1116 = 'Outputs'
  10548 = 'Outputs, PROFINET receive data'
  7984 = 'Outputs, PROFINET send data'
  797 = 'Overrange'
  291 = 'P'
  399 = 'p'
  1130 = 'P-Gain'
  7846 = 'P1'
  18520 = 'P2'
  16371 = 'P3'
  2574 = 'P4'
  667 = 'pA'
  1868 = 'PA'
  13235 = 'PA / PC sync after done'
  5492 = 'PA/PC sync after done'
  11770 = 'PA1 WorkerPos'
  875 = 'Paper Pos. Detction'
  709 = 'Park'
  4056 = 'ParkPosition'
  5893 = 'Pass Nb %d'
  6460 = 'Pass Nb: %d'
  7897 = 'PassNumber'
  2215 = 'PassOffset'
  3466 = 'Password'
  12139 = 'path name'
  3456 = "path to file location, needs an '\\' at the end of string"
  57 = 'Pattern'
  66 = 'Pattern: 0x%8.8x'
  348 = 'Pause'
  668 = 'pB'
  1218 = 'PC'
  385 = 'PC %d'
  229 = 'PC disabled!'
  356 = 'PC Index'
  7311 = 'PC range'
  369 = 'PC%s'
  345 = 'pCoeValue'
  384 = 'PC[ %d ]'
  237 = 'Per PH'
  764 = 'Period: %d [ms]'
  2720 = 'PG'
  190 = 'Pg cfg'
  12785 = 'PG enable'
  18326 = 'PG Enable'
  121 = 'PG Offset'
  436 = 'PG offset'
  186 = 'PG Offset\n(changeable dynamically)'
  455 = 'PG Offset [m]'
  173 = 'PG Shift'
  20065 = 'PG%d'
  500 = 'PG1'
  8391 = 'PG1 SubRow delta'
  501 = 'PG2'
  14461 = 'PG3'
  10402 = 'PG4'
  285 = 'PH'
  2432 = 'PH 1'
  2447 = 'PH 10'
  2449 = 'PH 11'
  7886 = 'PH 12'
  7891 = 'PH 13'
  7969 = 'PH 14'
  9042 = 'PH 15'
  7902 = 'PH 16'
  7907 = 'PH 17'
  7912 = 'PH 18'
  7917 = 'PH 19'
  2434 = 'PH 2'
  7923 = 'PH 20'
  7928 = 'PH 21'
  7933 = 'PH 22'
  7938 = 'PH 23'
  7943 = 'PH 24'
  7949 = 'PH 25'
  7954 = 'PH 26'
  7959 = 'PH 27'
  7964 = 'PH 28'
  5529 = 'PH 29'
  2436 = 'PH 3'
  11280 = 'PH 30'
  15501 = 'PH 31'
  5267 = 'PH 32'
  15875 = 'PH 33'
  2887 = 'PH 34'
  4096 = 'PH 35'
  9160 = 'PH 36'
  5864 = 'PH 37'
  4502 = 'PH 38'
  5558 = 'PH 39'
  2437 = 'PH 4'
  2944 = 'PH 40'
  2439 = 'PH 5'
  2441 = 'PH 6'
  2443 = 'PH 7'
  2445 = 'PH 8'
  2446 = 'PH 9'
  354 = 'PH Id'
  1652 = 'PH Master'
  873 = 'PH Master Setup'
  862 = 'PH Offset'
  802 = 'PH Offset [um]: %d'
  136 = 'PH Present'
  393 = 'PH Res.[dpi]'
  355 = 'PH Sel'
  6012 = 'PH Setup'
  394 = 'PH SubPx'
  18180 = 'PH%d'
  16887 = 'PH%s'
  15654 = 'PhMaster FilterDepth'
  159 = 'PH[%d]'
  2703 = 'Pinning closed'
  1125 = 'Pinning not closed'
  3487 = 'Pinning Start Offset'
  4832 = 'Pinning state'
  4415 = 'Pinning StopMargin'
  676 = 'Place'
  728 = 'PLC Settings'
  479 = 'PLC Status'
  14670 = 'PM'
  18128 = 'PM Detail'
  1648 = 'PM Master'
  20782 = 'PM Y adjust [µm]'
  13698 = 'PM1'
  9706 = 'PM2'
  16202 = 'PM: %d'
  526 = 'Port State'
  21704 = 'Pos'
  7539 = 'pos x [cm]'
  435 = 'Pos X0'
  14528 = 'PosCylinderDiameter [mm]'
  396 = 'position'
  401 = 'Position'
  16820 = 'Position --> Motion'
  3807 = 'Position A'
  2199 = 'Position B'
  680 = 'Position p1'
  681 = 'Position p2'
  3858 = 'Position [mm]'
  392 = 'PositionMaster: %d '
  682 = 'POSITIONS'
  888 = 'Positions'
  2355 = 'PositionShift'
  13394 = 'Power Hw ON'
  149 = 'Preparing'
  418 = 'PrePostBlank'
  429 = 'PrePostDepth'
  2051 = 'Press act back'
  301 = 'Press Act Val'
  1173 = 'Press actual'
  1175 = 'Press actual [mbar]'
  3020 = 'Press Delta'
  1174 = 'Press delta [mbar]'
  302 = 'Press Set Val'
  4686 = 'Press target'
  11824 = 'Press target  [mbar]'
  7667 = 'Press target [mbar]'
  300 = 'PressMinus'
  312 = 'PressPlus'
  1054 = 'pressure feedback'
  1049 = 'Pressure generation'
  1055 = 'pressure set point'
  1056 = 'pressure setpoint'
  1048 = 'pressure setpoint %1.1f [V]'
  1051 = 'Pressure setpoint %1.1f [V]'
  1047 = 'pressure setpoint [V]'
  1013 = 'pressure setting'
  1053 = 'Pressure setting'
  1014 = 'pressure setting\n[mbar]'
  1007 = 'PRG_ENABLING.iL_PressureSettingTable[0,INDEX]'
  1006 = 'PRG_ENABLING.iL_VarnishQuantityTable[INDEX]'
  1162 = 'PRG_INK.fR_HTFilterSupervisionPumpSpeed[1,INDEX]'
  9085 = 'PRG_INK.fR_HTFilterSupervisionPumpSpeed[INDEX1,INDEX2]'
  12417 = 'PRG_PRINT LogLevel'
  164 = 'Print'
  738 = 'Print '
  130 = 'Print Abort'
  14694 = 'Print Details'
  162 = 'Print enable'
  14325 = 'Print enabled'
  766 = 'Print maintenance image if invalid index is found: %d'
  51 = 'Print Mode : 0x%8.8x'
  870 = 'Print Motion Signals'
  169 = 'Print Pause'
  4799 = 'Print Pos'
  127 = 'Print Prepare'
  4782 = 'Print Speed'
  128 = 'Print Start'
  129 = 'Print Stop'
  734 = 'Print Unit'
  252 = 'Print Unit\nVISU_PU'
  4516 = 'Print unit (max %d)'
  1181 = 'Print1'
  18109 = 'Print2'
  4651 = 'Printed columns'
  43 = 'Printed Copies : %d'
  11865 = 'PrintEnabled'
  815 = 'Printer Ready'
  1184 = 'PrinterReady'
  5941 = 'PrintGroup: %d'
  141 = 'Printhead 1'
  287 = 'Printhead 1\n    (rear)'
  1081 = 'Printhead 1.1'
  1082 = 'Printhead 1.2'
  1083 = 'Printhead 1.3'
  1084 = 'Printhead 1.4'
  1085 = 'Printhead 1.5'
  1086 = 'Printhead 1.6'
  9499 = 'Printhead 1.7'
  1856 = 'Printhead 1.8'
  837 = 'Printhead 10'
  838 = 'Printhead 11'
  839 = 'Printhead 12'
  840 = 'Printhead 13'
  841 = 'Printhead 14'
  842 = 'Printhead 15'
  1005 = 'Printhead 15,'
  843 = 'Printhead 16'
  844 = 'Printhead 17'
  845 = 'Printhead 18'
  948 = 'Printhead 19'
  846 = 'Printhead 195'
  143 = 'Printhead 2'
  288 = 'Printhead 2\n  (center)'
  1087 = 'Printhead 2.1'
  1088 = 'Printhead 2.2'
  1089 = 'Printhead 2.3'
  1090 = 'Printhead 2.4'
  1091 = 'Printhead 2.5'
  1092 = 'Printhead 2.6'
  847 = 'Printhead 20'
  848 = 'Printhead 21'
  849 = 'Printhead 22'
  850 = 'Printhead 23'
  851 = 'Printhead 24'
  852 = 'Printhead 25'
  949 = 'Printhead 26'
  853 = 'Printhead 262'
  854 = 'Printhead 27'
  855 = 'Printhead 28'
  144 = 'Printhead 3'
  289 = 'Printhead 3\n   (front)'
  145 = 'Printhead 4'
  832 = 'Printhead 5'
  833 = 'Printhead 6'
  834 = 'Printhead 7'
  835 = 'Printhead 8'
  836 = 'Printhead 9'
  112 = 'Printhead Resolution'
  286 = 'Printhead selection\nfor purge'
  151 = 'Printing'
  431 = 'PrintLength'
  2760 = 'Printline 1'
  8759 = 'Printline 2'
  12243 = 'Printline 3'
  16572 = 'Printline 4'
  414 = 'PrintMode'
  3475 = 'PrintModule'
  5645 = 'PrintModule %d'
  1182 = 'PrintModule%d'
  1163 = 'PrintOffset [SubPx]:: %d'
  1536 = 'PrintPosition'
  3397 = 'PrintUnit'
  11391 = 'Process'
  426 = 'Prod.Images'
  897 = 'Product'
  5301 = 'ProductionSpeed'
  175 = 'Products'
  18003 = 'Profiler'
  225 = 'Progress'
  896 = 'Project'
  895 = 'Project Information'
  5878 = 'PU'
  15081 = 'PU Elevation'
  1198 = 'PU Elevation [m]'
  16528 = 'PU in position'
  158 = 'Pulse'
  439 = 'Pulse duration'
  157 = 'PULSE GENERATOR'
  257 = 'Pump'
  997 = 'Pump %'
  516 = 'Pump Activated'
  1701 = 'Pump active'
  4191 = 'Pump cycle'
  9806 = 'Pump speed'
  282 = 'Pump time too long\n Tank is not filled?'
  575 = 'PUMPE'
  283 = 'Purge'
  600 = 'PURGE'
  604 = 'Purge active station'
  721 = 'Purge after Capping'
  12482 = 'Purge conditions'
  325 = 'Purge controller %s'
  1142 = 'Purge controller groups'
  324 = 'Purge cycle'
  614 = 'PURGE CYCLE'
  8643 = 'Purge machine conditions'
  610 = 'PURGE REPEATS'
  284 = 'Purge selected'
  1724 = 'Purge selection'
  8401 = 'Purge sequence'
  1143 = 'Purge sequence DSU'
  615 = 'PURGE SETTINGS'
  596 = 'Purge should be activated\nmanually after exchange'
  608 = 'PURGE TIME'
  323 = 'Purge time total'
  613 = 'Purge Time Total'
  601 = 'Purge Ventil'
  609 = 'PURGE WAIT TIME'
  188 = 'px: %d'
  8246 = 'Qualivision line camera'
  359 = 'Queue'
  137 = 'Queue empty'
  378 = 'queue full'
  90 = 'R'
  644 = 'RAMP'
  1031 = 'range [mbar]\ngap [0.1mm]\ntemperature [0.1°C'
  1032 = 'range [mbar]\ngap [0.1mm]\ntemperature [0.1°C]'
  9886 = 'Rated Capacity (Emax):'
  13237 = 'Rated Output (Cn):'
  453 = 'RdIdx'
  347 = 'RdReq'
  202 = 'Read'
  41 = 'Read Status'
  443 = 'ReadCond.'
  13731 = 'Readings'
  351 = 'ReadReq'
  150 = 'Ready'
  458 = 'Ready:'
  4175 = 'Rec count'
  537 = 'Receive Frame'
  4137 = 'Receive test'
  7235 = 'Recipe'
  753 = 'Reconnect'
  703 = 'Ref'
  15190 = 'REF Master'
  4791 = 'Ref Pos'
  4774 = 'Ref Speed'
  6747 = 'Reference Weight:'
  9362 = 'RefMaster FilterDepth'
  468 = 'Refresh'
  29 = 'Refresh Rate'
  580 = 'REFUSE'
  249 = 'Refuse / Exchange / Cleaner\nVISU_MAINTENANCE'
  566 = 'REFUSE / EXCHANGE VARNISH'
  597 = 'Refuse delay ink pump'
  598 = 'Refuse time ink pump'
  1172 = 'Refuse to storage tank'
  628 = 'REFUSE VARNISH PUMP'
  568 = 'Refuse-'
  364 = 'Reg: %d'
  672 = 'RegActive'
  16819 = 'Register Mark'
  45 = 'Register new Job'
  86 = 'REM'
  16 = 'Rem. Time'
  87 = 'remove'
  486 = 'Remove Job'
  331 = 'Reopen\nvalves at\npressure\nPx'
  77 = 'Repeat'
  2586 = 'Reset'
  91 = 'Reset board'
  810 = 'Reset FB PaperDet.'
  811 = 'Reset FB Ringbuffer'
  2241 = 'Reset filter was changed'
  11211 = 'Reset last scanned entry'
  107 = 'Reset PHMaster'
  960 = 'Reset state machine'
  959 = 'Reset statemachine'
  8560 = 'Reset test'
  1151 = 'Reset, filter was changed'
  787 = 'Resolution'
  47 = 'Resolution : %d'
  428 = 'ResolutionX'
  752 = 'Response'
  349 = 'Retries'
  9760 = 'Return flow measurement'
  950 = 'Return flow time'
  951 = 'Return flow time [s]'
  877 = 'Ringbuffer Elements'
  433 = 'RingBuffer: %d '
  11409 = 'Roll table'
  2537 = 'Roll table (max %d)'
  10338 = 'RT circulation pump'
  2247 = 'RT diameter'
  1140 = 'RT diameter [mm]'
  2675 = 'RT fill pump supervision'
  6695 = 'RT long [°C]'
  1723 = 'RT short [°C]'
  5460 = 'RT test amount [cm³/min]'
  6072 = 'RT test amount [mm³/min]'
  4445 = 'Run down delay'
  3142 = 'Running'
  2823 = 'rx'
  2076 = 'ry'
  407 = 'S'
  695 = 'Safe Running Condition'
  692 = 'Safety'
  17962 = 'Safety cover'
  1065 = 'safety distance'
  15672 = 'Safety doors'
  8652 = 'Safety ok'
  690 = 'SafetyConditionOK'
  4144 = 'Scan state'
  4125 = 'Scanned label false!'
  4118 = 'Scanned tank ID'
  11691 = 'SD'
  1192 = 'sdf'
  789 = 'Segment Count'
  794 = 'Segment Index'
  788 = 'Segment Size'
  790 = 'SegmentAngle'
  78 = 'Segmented'
  430 = 'SegmentLength'
  7047 = 'Sel PH : %d '
  561 = 'SEL TANK'
  15622 = 'select'
  477 = 'Select Folder'
  595 = 'Select headertank (multiple)'
  588 = 'Select headertank (only one)'
  584 = 'Select headertank for auto (only one)'
  478 = 'Select Image'
  1188 = 'select inverted'
  6169 = 'select normal'
  292 = 'Select purge'
  589 = 'Select tank'
  599 = 'SEL_PURGE'
  520 = 'Send Frame'
  55 = 'Send Job Cmd'
  65 = 'SendCommand'
  578 = 'SENSOR'
  264 = 'Sensor (full)'
  830 = 'Sensor S1-S2'
  3927 = 'Seperator niveau'
  742 = 'Serv'
  678 = 'Service'
  1076 = 'Service / DEM not engage'
  1077 = 'Service / DEM not engaged'
  3928 = 'SERVICE White'
  688 = 'ServiceEnabled'
  167 = 'SERVICES'
  4356 = 'Set'
  3684 = 'Set  Tara'
  9057 = 'Set nb passes: %d'
  6901 = 'Set nb steps: %d'
  11540 = 'Set RefWeght'
  11474 = 'Set RefWeight'
  6512 = 'Set steps: %d'
  297 = 'Set Value in [%s]'
  309 = 'Set Value in [mbar]'
  3133 = 'Set YOffset: %d'
  13297 = 'Set YOffset: %d [px]'
  12847 = 'Set Zero'
  739 = 'Set:10'
  5081 = 'Setpoint #1 [%]'
  2548 = 'Setpoint #2 [%]'
  1673 = 'Setpoint #3 [%]'
  3808 = 'Setpoint #4 [%]'
  2275 = 'Setpoint intensity'
  258 = 'Setpoint pump'
  582 = 'SETPOINT PUMP %'
  624 = 'SETPOINT REFUSE PUMP %'
  662 = 'SETPOINT TEMP CALC [0.1°C]'
  936 = 'Setpoint temp calc [0.1°C]'
  654 = 'SETPOINT TEMP [°C]'
  937 = 'Setpoint temp [°C]'
  6231 = 'SETTING'
  61 = 'Settings'
  630 = 'Settings Cleaner pump '
  9094 = 'Settings Cleaner pump cleaning station'
  4826 = 'Settings Cleaner pump headertank'
  276 = 'Settings fill ink pump %s'
  11046 = 'Settings Fill pump'
  631 = 'Settings Fill pump VARNISH'
  635 = 'Settings ramp for fill pump VARNISH'
  627 = 'Settings Refuse pump VARNISH'
  641 = 'Settings temp controller HT'
  639 = 'Settings temp controller PH'
  340 = 'Settings unfill ink pump %s'
  4706 = 'Settings WEU'
  769 = 'Settings with (X) must be enabled to simulate a multipage job'
  14005 = 'Setup'
  6153 = 'Setup SpeedCompensation'
  31 = 'Set_Zero'
  2719 = 'sfd'
  809 = 'Sheet Angle'
  813 = 'Sheet y Offset'
  2258 = 'SheetCycle'
  1382 = 'SheetDetect'
  3305 = 'SheetGap'
  1161 = 'SheetLength'
  2238 = 'SheetTrigger'
  201 = 'Shift'
  449 = 'Shift distance'
  8377 = 'Shift start correction'
  988 = 'Shift start correction:'
  5168 = 'ShiftFact'
  6358 = 'ShiftOffs'
  371 = 'Show details'
  6611 = 'Show Details'
  21803 = 'Show PC'
  2732 = 'Show PC: %d'
  20887 = 'Show PH'
  17493 = 'Show PH %d'
  10534 = 'Show PH: %d'
  727 = 'Shutter'
  751 = 'SICK AG'
  1778 = 'Sim Encoder (all)'
  9081 = 'Sim Engage'
  17253 = 'Sim format (cyclic)'
  1951 = 'Sim GridPoint on PH[1]'
  11971 = 'Sim Machine Ready'
  18626 = 'Sim MarkDetection'
  8475 = 'Sim Master Positions (all)'
  2650 = 'Sim PhMaster'
  10878 = 'Sim PhMaster M2: %0.2f [m/s]'
  16553 = 'Sim PhMaster M3: %0.2f [m/s]'
  12848 = 'Sim PhMaster: %0.2f [m/s]'
  5898 = 'Sim position'
  2393 = 'Sim Position %0.3f [m/s]'
  15777 = 'Sim Position %f [m/s]'
  16743 = 'Sim position (all)'
  11131 = 'Sim PRG_INK'
  3415 = 'Sim PRG_MACHINE'
  16986 = 'Sim PRG_PRINT'
  9089 = 'Sim PrintEnable'
  9379 = 'Sim Sheets (cyclic)'
  1255 = 'Sim StartTrigger (cyclic)'
  12357 = 'Sim VEncoder'
  16679 = 'sImgId'
  5384 = 'SimSpeed'
  122 = 'Simulate'
  11236 = 'Simulation'
  768 = 'Simulation (X)'
  19416 = 'Simulation mode'
  126 = 'Slave Addr'
  9107 = 'Sleep'
  564 = 'Sleep active'
  11570 = 'Sleep active, sleep command'
  5060 = 'Slot1'
  1169 = 'Slot10'
  11794 = 'Slot2'
  2311 = 'Slot3'
  5977 = 'Slot4'
  9612 = 'Slot5'
  2811 = 'Slot6'
  5615 = 'Slot7'
  1166 = 'Slot8'
  1168 = 'Slot9'
  7005 = 'Smulation'
  230 = 'Some PC in range are \nnot enabled!'
  7318 = 'Some PC in range are \nNOT enabled!'
  2523 = 'Some VISUs '
  60 = 'Source'
  3460 = 'SourcePath'
  269 = 'Speed'
  12744 = 'Speed >5m/min'
  15504 = 'Speed m/min'
  181 = 'Speed m/s'
  6494 = 'Speed Module2'
  1359 = 'Speed Module2 [m/min]'
  5595 = 'Speed Module3'
  16486 = 'Speed Module3 [m/min]'
  2930 = 'Speed valid'
  9942 = 'Speed [%]'
  15688 = 'Speed [m/min]'
  9363 = 'Speed [m/s]'
  1124 = 'Speed [m/s]: %f'
  3084 = 'SpeedComp'
  863 = 'SpeedCompensation'
  18209 = 'SpeedExeeded'
  674 = 'SPEEDS'
  95 = 'Spit cmd state'
  101 = 'Spit Data'
  100 = 'Spit Frequency [kHz]'
  92 = 'Spitting manual'
  1063 = 'Splice detection: enable'
  4565 = 'sq: %0.3f'
  12942 = 'sq:%0.3f'
  10101 = 'sState'
  11 = 'ST Act Level'
  12 = 'ST Status'
  4781 = 'Standby'
  235 = 'Start'
  6070 = 'Start (manual)'
  218 = 'Start ALL'
  712 = 'Start Cleaning'
  924 = 'Start Empty'
  3447 = 'Start file download'
  925 = 'Start Fill'
  919 = 'Start Flush'
  7605 = 'Start HIB Update'
  767 = 'Start index: %d'
  1871 = 'Start Job'
  883 = 'Start Pos. Correction'
  713 = 'Start Purge'
  170 = 'Start Trigger'
  4358 = 'Start up offset'
  445 = 'Start XO'
  446 = 'Start XS'
  7082 = 'StartCanEx'
  8070 = 'Started'
  1480 = 'StartExec'
  14907 = 'Starting'
  1620 = 'StartOffs'
  9704 = 'StartPosDetect'
  11923 = 'StartTrigger'
  756 = 'StartTriggerTest'
  148 = 'STATE'
  176 = 'State'
  6119 = 'state'
  7434 = 'State name'
  7562 = 'Statemachine State'
  780 = 'Static Angle Offset'
  792 = 'Static Y Offset'
  18 = 'Status'
  507 = 'STATUS'
  42 = 'Status : 0x%8.8x'
  11686 = 'Stop (manual)'
  1926 = 'Stop cleaner'
  8213 = 'Stop flushing cycle'
  3474 = 'Stop Job'
  172 = 'Stop Trigger'
  7189 = 'StopCanEx'
  9543 = 'StopExec'
  15149 = 'Stopping'
  7154 = 'STORAGE'
  10427 = 'Storage container AdsID actual value'
  5 = 'Storage Tank'
  562 = 'STORAGE TANK'
  10995 = 'Storage tank %s ID'
  963 = 'Storage tank 1 assignment ID'
  964 = 'Storage tank 2 assignment ID'
  13957 = 'Storage tank 3 assignment ID'
  8119 = 'Storage tank 4 assignment ID'
  7326 = 'Storage tank 5 assignment ID'
  931 = 'Storage tank assignment actual value'
  930 = 'Storage tank assignment set value'
  280 = 'Sub\nmeniscus'
  7911 = 'Sub menc factor'
  2407 = 'Sub menc factor [%]'
  7937 = 'Sub menc neg factor [%]'
  12519 = 'Sub menc neg ramp [s]'
  5905 = 'Sub menc pos factor [%]'
  10336 = 'Sub menc pos ramp'
  2225 = 'Sub menc pos ramp [s]'
  906 = 'Sub meniscus'
  205 = 'Subindex'
  996 = 'SubMenc'
  335 = 'SubMenc %s'
  15303 = 'SubMenc1 adjust Purge/Clean'
  14324 = 'SubMenc2 adjust Purge/Clean'
  402 = 'SubPixel-'
  806 = 'Substrate Length'
  7470 = 'Substrate thickness [m]: %f'
  3446 = 'SubstrateLength'
  1519 = 'SubstrateLength effect.'
  13585 = 'SubstrateThickness'
  16704 = 'SubstrateThickness [µm]'
  14279 = 'SubstrateWidth'
  872 = 'SubtrateLength [m] : %f'
  377 = 'success'
  10926 = 'Supervision relay'
  11935 = 'Supervision window'
  114 = 'SupPixel Resolution'
  131 = 'Sync'
  139 = 'Sync Warning'
  515 = 'SYSTEM'
  6017 = 'System'
  687 = 'SystemReady'
  8252 = 'Systron camera'
  770 = 'systron GmbH'
  437 = 'T'
  338 = 'T delay off'
  339 = 'T delay on'
  594 = 'T Exchange interval'
  647 = 'T max'
  918 = 'T max active'
  607 = 'T max Manu'
  326 = 'T maxTest'
  274 = 'T pump off'
  587 = 'T Refuse / Exchange'
  14239 = 'T return flow'
  275 = 'T valve on'
  316 = 'T Wait Manu'
  10620 = 'Table'
  4275 = 'Table set counter value: %d'
  571 = 'tank'
  602 = 'Tank 1'
  616 = 'Tank 2'
  617 = 'Tank 3'
  995 = 'Tank 4'
  618 = 'Tank 5'
  619 = 'Tank 6'
  620 = 'Tank 7'
  23 = 'Tank Size'
  6200 = 'Tare Weight:'
  700 = 'Target'
  5478 = 'Target speed reached'
  11241 = 'TcpIpClient'
  15269 = 'teached marks'
  8677 = 'TEMP'
  13839 = 'TEMP CMYK'
  643 = 'TEMP Header-Tank'
  640 = 'TEMP Print-Head plate'
  1170 = 'TEMP W'
  6029 = 'TEMP White'
  198 = 'Temperature'
  1060 = 'Temperature feedback'
  1062 = 'temperature setpoint'
  1061 = 'temperature teedback'
  62 = 'Test'
  298 = 'Test (=Contr Off)'
  5855 = 'Test active'
  1571 = 'Test amount [cm³/min]'
  5705 = 'Test amount [cm³]'
  3943 = 'test amount [mm^3]'
  11248 = 'Test amount [mm³/min]'
  1147 = 'Test amount [mm³/s]'
  2350 = 'test amount [mm³]'
  7394 = 'Test amount [mm³]'
  3160 = 'Test balance'
  5578 = 'Test interval'
  17621 = 'Test mark 1'
  9550 = 'Test mark 2'
  14487 = 'Test Mmark 1'
  308 = 'Test Off'
  307 = 'Test Press Minus'
  311 = 'Test Press Plus'
  4794 = 'Test start'
  8300 = 'Test time'
  8226 = 'TEST01'
  1251 = 'Test1'
  2109 = 'Test2'
  755 = 'Test: NewValue'
  8409 = 'Testing'
  13578 = 'Testing & Simulation'
  9047 = 'Testing initialized'
  14062 = 'TestJob'
  5287 = 'Time'
  5511 = 'Time after BiB change'
  6047 = 'Time after Purge'
  952 = 'Time blow out [s]'
  954 = 'Time empty cleaner [s]'
  1127 = 'Time Mark-Mark'
  10818 = 'Time menc ok'
  5722 = 'Time no movement'
  4285 = 'Time re check detector'
  9103 = 'Time recheck detector'
  16021 = 'Time refuse flow [s]'
  13274 = 'Time resume circ.'
  953 = 'Time return flow [s]'
  634 = 'time s'
  4901 = 'Time separator pump for tank drainage'
  955 = 'Time warn exchange [h]'
  1159 = 'Time [ms]: %d'
  12547 = 'Time [ms]: %s'
  9795 = 'Time [ms]: %t'
  9575 = 'Timeout after: %s'
  637 = 'timer'
  910 = 'Timer'
  380 = 'Timestamp'
  227 = 'To      PC:'
  191 = 'To PCs'
  14553 = 'TODO'
  11635 = 'TODO add ALL Persistent Values!!!!'
  305 = 'Tol Wdw big'
  304 = 'Tol Wdw small'
  19257 = 'Tolerance'
  5291 = 'Tolerance for compare sheet length with image depth'
  3764 = 'Tool Selection'
  5716 = 'Total columns'
  19513 = 'tr: %0.3f'
  7951 = 'tr:%0.3f'
  5292 = 'TrackPos'
  165 = 'Transfer'
  138 = 'Transfer active'
  475 = 'Transfer Complete'
  480 = 'Transfer Error'
  481 = 'Transfer Go'
  214 = 'Transfer size'
  814 = 'Transport Ready'
  438 = 'Trigger'
  7998 = 'Trigger active'
  7753 = 'Trigger Armed'
  8586 = 'Trigger distance'
  777 = 'Trigger Generation'
  763 = 'Trigger generator'
  233 = 'Trigger manual update'
  4420 = 'Trigger pulse length'
  773 = 'TriggerFeedback'
  13192 = 'TrigToCam'
  466 = 'Type:'
  8274 = 'UDP receive data'
  8202 = 'UDP send data'
  400 = 'um'
  4710 = 'um: %d'
  796 = 'Underrange'
  670 = 'UNDO'
  278 = 'Unfill'
  337 = 'Unfill %s'
  592 = 'Unit not in capping mode!'
  224 = 'Unlock Patern'
  958 = 'Unlock Pattern'
  957 = 'Unlock Reset'
  223 = 'Update FPGA on all enabled Boards'
  7598 = 'Update FSM  of selected PC'
  221 = 'Update FW on all enabled Boards'
  7591 = 'USAGE:\nEnter password, set PC range, start HIB Update\n\nNOTE:\nUpdate HAB firmware only if no waveform download is active on the selected ControllerBoards!!!\nCheck version after download!\n\nThis feature works, but is in Beta state. Implementation, Visualisation and usage will change.'
  867 = 'Use AuxEncoder'
  771 = 'Use camera system'
  240 = 'Use default file'
  3453 = 'Use default file: %s'
  6272 = 'Use Enc C emulation (instead of Marks)'
  15390 = 'Use EncoderC instead of Marks'
  11014 = 'Use EncoderC instead of marks'
  12500 = 'Use EncoderC instead of Markus'
  759 = 'Use scanner index for image offset (X)'
  5948 = 'V'
  5809 = 'VACUUM'
  1189 = 'Vacuum FU error'
  4759 = 'Vacuum pump'
  7471 = 'Vacuum pump activation'
  649 = 'Vacuum pump max time'
  9833 = 'Vacuum warn/err'
  14190 = 'Vacuum warn/error'
  263 = 'Valve'
  576 = 'VALVE'
  912 = 'Varnish density'
  904 = 'Varnish parameter'
  1012 = 'varnish quantity [g/m2]'
  914 = 'Varnish viscosity'
  4250 = 'VD'
  19446 = 'Verbose'
  3014 = 'Verbose Mode'
  898 = 'Version'
  461 = 'Version:'
  452 = 'vGap'
  8797 = 'View MarkScale'
  881 = 'Virtual StartShift Group1'
  882 = 'Virtual StartShift Group2'
  246 = 'VISU_ADS_INKSTORAGE_TANK'
  242 = 'VISU_INK'
  7006 = 'VISU_PRINT'
  251 = 'VISU_PROCESS'
  243 = 'VISU_PURGE'
  250 = 'VISU_SETTINGS'
  3051 = 'VISU_SYSTEMBASE'
  908 = 'Voltage scaling'
  803 = 'vShift start [m] : %f'
  874 = 'vShift_G1 start [m] : %f'
  1119 = 'vShift_G1 [m] : %f'
  876 = 'vShift_G2 start [m] : %f'
  1120 = 'vShift_G2 [m] : %f'
  547 = 'VT_1.01'
  998 = 'VT_1.02'
  549 = 'VT_1.06'
  1071 = 'VT_1.1'
  551 = 'VT_1.11'
  1074 = 'VT_1.2'
  553 = 'VT_2.01'
  1000 = 'VT_2.02'
  999 = 'VT_2.03'
  555 = 'VT_2.06'
  1072 = 'VT_2.1'
  557 = 'VT_2.11'
  1073 = 'VT_2.2'
  3123 = 'W'
  745 = 'Wait'
  15170 = 'Wait start: %s'
  334 = 'Wait time'
  611 = 'WAIT VALVE ON'
  374 = 'waiting'
  746 = 'Waiting'
  8962 = 'Wake up'
  14291 = 'WakeUp'
  5313 = 'wakeup command'
  133 = 'Warning'
  4224 = 'Warning level'
  19708 = 'Warning Message active'
